LIN {X 0,Y 411.201,Z 268.89,A -85,B 0,C 180,E1 -10404.471,E2 -10404.471} C_VEL
LIN {X 0,Y 411.211,Z 268.89,A -85,B 0,C 180,E1 -10406.873,E2 -10406.873} C_VEL
LIN {X 0,Y 411.237,Z 268.886,A -85,B 0,C 180,E1 -10410.644,E2 -10410.644} C_VEL
LIN {X 0,Y 411.238,Z 268.882,A -85,B 0,C 180,E1 -10413.619,E2 -10413.619} C_VEL
LIN {X 0,Y 411.2,Z 268.891,A -85,B 0,C 180,E1 -10416.852,E2 -10416.852} C_VEL
LIN {X 0,Y 411.219,Z 268.887,A -85,B 0,C 180,E1 -10420.05,E2 -10420.05} C_VEL
LIN {X 0,Y 411.268,Z 268.88,A -85,B 0,C 180,E1 -10423.131,E2 -10423.131} C_VEL
LIN {X 0,Y 411.31,Z 268.874,A -85,B 0,C 180,E1 -10426.896,E2 -10426.896} C_VEL
LIN {X 0,Y 411.296,Z 268.879,A -85,B 0,C 180,E1 -10430.161,E2 -10430.161} C_VEL
LIN {X 0,Y 411.395,Z 268.863,A -85,B 0,C 180,E1 -10433.132,E2 -10433.132} C_VEL
LIN {X 0,Y 411.302,Z 268.875,A -85,B 0,C 180,E1 -10435.099,E2 -10435.099} C_VEL
LIN {X 0,Y 411.515,Z 268.851,A -85,B 0,C 180,E1 -10438.042,E2 -10438.042} C_VEL
LIN {X 0,Y 411.638,Z 268.837,A -85,B 0,C 180,E1 -10440,E2 -10440} C_VEL
LIN {X 0,Y 411.462,Z 268.856,A -85,B 0,C 180,E1 -10442.937,E2 -10442.937} C_VEL
LIN {X 0,Y 411.441,Z 268.861,A -85,B 0,C 180,E1 -10445.882,E2 -10445.882} C_VEL
LIN {X 0,Y 411.321,Z 268.872,A -85,B 0,C 180,E1 -10448.846,E2 -10448.846} C_VEL
LIN {X 0,Y 411.287,Z 268.88,A -85,B 0,C 180,E1 -10451.832,E2 -10451.832} C_VEL
LIN {X 0,Y 411.262,Z 268.879,A -85,B 0,C 180,E1 -10454.852,E2 -10454.852} C_VEL
LIN {X 0,Y 411.254,Z 268.884,A -85,B 0,C 180,E1 -10457.915,E2 -10457.915} C_VEL
LIN {X 0,Y 411.2,Z 268.889,A -85,B 0,C 180,E1 -10461.034,E2 -10461.034} C_VEL
LIN {X 0,Y 411.221,Z 268.886,A -85,B 0,C 180,E1 -10464.216,E2 -10464.216} C_VEL
LIN {X 0,Y 411.181,Z 268.895,A -85,B 0,C 180,E1 -10467.483,E2 -10467.483} C_VEL
LIN {X 0,Y 411.199,Z 268.89,A -85,B 0,C 180,E1 -10469.713,E2 -10469.713} C_VEL
LIN {X 0,Y 411.209,Z 268.89,A -85,B 0,C 180,E1 -10473.155,E2 -10473.155} C_VEL
LIN {X 0,Y 411.194,Z 268.889,A -85,B 0,C 180,E1 -10476.552,E2 -10476.552} C_VEL
LIN {X 0,Y 411.212,Z 268.897,A -85,B 0,C 180,E1 -10477.046,E2 -10477.046} C_VEL
LIN {X 0,Y 412.12,Z 274.033,A -85,B 0,C 180,E1 -10480.393,E2 -10480.393} C_VEL
LIN {X 0,Y 413.062,Z 279.177,A -85,B 0,C 180,E1 -10483.557,E2 -10483.557} C_VEL
LIN {X 0,Y 413.812,Z 283.108,A -85,B 0,C 180,E1 -10485.867,E2 -10485.867} C_VEL
LIN {X 0,Y 414.18,Z 285.575,A -85,B 0,C 180,E1 -10487.254,E2 -10487.254} C_VEL
LIN {X 0,Y 414.126,Z 289.23,A -85,B 0,C 180,E1 -10489.204,E2 -10489.204} C_VEL
LIN {X 0,Y 413.62,Z 295.329,A -85,B 0,C 180,E1 -10492.288,E2 -10492.288} C_VEL
LIN {X 0,Y 412.949,Z 302.639,A -85,B 0,C 180,E1 -10495.831,E2 -10495.831} C_VEL
LIN {X 0,Y 412.403,Z 309.967,A -85,B 0,C 180,E1 -10499.253,E2 -10499.253} C_VEL
LIN {X 0,Y 411.862,Z 317.318,A -85,B 0,C 180,E1 -10502.566,E2 -10502.566} C_VEL
LIN {X 0,Y 411.503,Z 322.706,A -85,B 0,C 180,E1 -10504.939,E2 -10504.939} C_VEL
LIN {X 0,Y 416.225,Z 340.747,A -85,B 0,C 180,E1 -10505.754,E2 -10505.754} C_VEL
LIN {X 0,Y 419.587,Z 356.286,A -85,B 0,C 180,E1 -10506.607,E2 -10506.607} C_VEL
LIN {X 0,Y 420.32,Z 360.595,A -85,B 0,C 180,E1 -10506.872,E2 -10506.872} C_VEL
LIN {X 0,Y 419.211,Z 375.514,A -85,B 0,C 180,E1 -10507.709,E2 -10507.709} C_VEL
LIN {X 0,Y 417.84,Z 389.213,A -85,B 0,C 180,E1 -10508.67,E2 -10508.67} C_VEL
LIN {X 0,Y 416.464,Z 403.182,A -85,B 0,C 180,E1 -10509.889,E2 -10509.889} C_VEL
LIN {X 0,Y 415.124,Z 415.883,A -85,B 0,C 180,E1 -10511.236,E2 -10511.236} C_VEL
LIN {X 0,Y 413.929,Z 427.487,A -85,B 0,C 180,E1 -10512.715,E2 -10512.715} C_VEL
LIN {X 0,Y 412.908,Z 437.298,A -85,B 0,C 180,E1 -10514.197,E2 -10514.197} C_VEL
LIN {X 0,Y 411.877,Z 446.94,A -85,B 0,C 180,E1 -10515.927,E2 -10515.927} C_VEL
LIN {X 0,Y 411.227,Z 455.004,A -85,B 0,C 180,E1 -10517.665,E2 -10517.665} C_VEL
LIN {X 0,Y 410.756,Z 460.8,A -85,B 0,C 180,E1 -10519.152,E2 -10519.152} C_VEL
LIN {X 0,Y 410.323,Z 467.138,A -85,B 0,C 180,E1 -10521.132,E2 -10521.132} C_VEL
LIN {X 0,Y 410.085,Z 472.043,A -85,B 0,C 180,E1 -10523.11,E2 -10523.11} C_VEL
LIN {X 0,Y 409.996,Z 475.633,A -85,B 0,C 180,E1 -10525.083,E2 -10525.083} C_VEL
LIN {X 0,Y 409.969,Z 477.983,A -85,B 0,C 180,E1 -10527.052,E2 -10527.052} C_VEL
LIN {X 0,Y 409.915,Z 479.141,A -85,B 0,C 180,E1 -10529.018,E2 -10529.018} C_VEL
LIN {X 0,Y 409.915,Z 479.086,A -85,B 0,C 180,E1 -10530.982,E2 -10530.982} C_VEL
LIN {X 0,Y 409.985,Z 477.829,A -85,B 0,C 180,E1 -10532.948,E2 -10532.948} C_VEL
LIN {X 0,Y 410.028,Z 475.37,A -85,B 0,C 180,E1 -10534.916,E2 -10534.916} C_VEL
LIN {X 0,Y 410.157,Z 471.659,A -85,B 0,C 180,E1 -10536.889,E2 -10536.889} C_VEL
LIN {X 0,Y 410.323,Z 466.595,A -85,B 0,C 180,E1 -10538.868,E2 -10538.868} C_VEL
LIN {X 0,Y 410.753,Z 460.062,A -85,B 0,C 180,E1 -10540.848,E2 -10540.848} C_VEL
LIN {X 0,Y 411.305,Z 451.879,A -85,B 0,C 180,E1 -10542.834,E2 -10542.834} C_VEL
LIN {X 0,Y 412.101,Z 443.193,A -85,B 0,C 180,E1 -10544.569,E2 -10544.569} C_VEL
LIN {X 0,Y 413.088,Z 432.798,A -85,B 0,C 180,E1 -10546.303,E2 -10546.303} C_VEL
LIN {X 0,Y 414.152,Z 422.254,A -85,B 0,C 180,E1 -10547.786,E2 -10547.786} C_VEL
LIN {X 0,Y 415.43,Z 409.781,A -85,B 0,C 180,E1 -10549.262,E2 -10549.262} C_VEL
LIN {X 0,Y 416.906,Z 396.092,A -85,B 0,C 180,E1 -10550.604,E2 -10550.604} C_VEL
LIN {X 0,Y 418.219,Z 382.713,A -85,B 0,C 180,E1 -10551.697,E2 -10551.697} C_VEL
LIN {X 0,Y 419.634,Z 367.281,A -85,B 0,C 180,E1 -10552.719,E2 -10552.719} C_VEL
LIN {X 0,Y 420.195,Z 359.819,A -85,B 0,C 180,E1 -10553.139,E2 -10553.139} C_VEL
LIN {X 0,Y 416.862,Z 341.94,A -85,B 0,C 180,E1 -10554.264,E2 -10554.264} C_VEL
LIN {X 0,Y 413.724,Z 327.801,A -85,B 0,C 180,E1 -10555.054,E2 -10555.054} C_VEL
LIN {X 0,Y 411.367,Z 319.22,A -85,B 0,C 180,E1 -10555.531,E2 -10555.531} C_VEL
LIN {X 0,Y 411.324,Z 318.857,A -85,B 0,C 180,E1 -10555.558,E2 -10555.558} C_VEL
LIN {X 0,Y 411.791,Z 310.923,A -85,B 0,C 180,E1 -10559.035,E2 -10559.035} C_VEL
LIN {X 0,Y 412.204,Z 304.79,A -85,B 0,C 180,E1 -10561.907,E2 -10561.907} C_VEL
LIN {X 0,Y 412.598,Z 300.233,A -85,B 0,C 180,E1 -10564.202,E2 -10564.202} C_VEL
LIN {X 0,Y 413.181,Z 295.3,A -85,B 0,C 180,E1 -10566.923,E2 -10566.923} C_VEL
LIN {X 0,Y 413.606,Z 292.035,A -85,B 0,C 180,E1 -10568.955,E2 -10568.955} C_VEL
LIN {X 0,Y 414.122,Z 288.293,A -85,B 0,C 180,E1 -10571.693,E2 -10571.693} C_VEL
LIN {X 0,Y 414.188,Z 286.686,A -85,B 0,C 180,E1 -10573.145,E2 -10573.145} C_VEL
LIN {X 0,Y 413.862,Z 284.426,A -85,B 0,C 180,E1 -10575.874,E2 -10575.874} C_VEL
LIN {X 0,Y 413.339,Z 283.119,A -85,B 0,C 180,E1 -10578.462,E2 -10578.462} C_VEL
LIN {X 0,Y 412.687,Z 282.48,A -85,B 0,C 180,E1 -10581.571,E2 -10581.571} C_VEL
LIN {X 0,Y 412.117,Z 282.678,A -85,B 0,C 180,E1 -10584.942,E2 -10584.942} C_VEL
LIN {X 0,Y 411.744,Z 283.465,A -85,B 0,C 180,E1 -10588.053,E2 -10588.053} C_VEL
LIN {X 0,Y 411.505,Z 284.692,A -85,B 0,C 180,E1 -10590.943,E2 -10590.943} C_VEL
LIN {X 0,Y 412.791,Z 287.703,A -85,B 0,C 180,E1 -10591.185,E2 -10591.185} C_VEL
LIN {X 0,Y 417.521,Z 298.226,A -85,B 0,C 180,E1 -10592.052,E2 -10592.052} C_VEL
LIN {X 0,Y 420.696,Z 307.253,A -85,B 0,C 180,E1 -10592.755,E2 -10592.755} C_VEL
LIN {X 0,Y 421.109,Z 308.983,A -85,B 0,C 180,E1 -10592.883,E2 -10592.883} C_VEL
LIN {X 0,Y 419.888,Z 325.497,A -85,B 0,C 180,E1 -10593.81,E2 -10593.81} C_VEL
LIN {X 0,Y 418.719,Z 339.594,A -85,B 0,C 180,E1 -10594.806,E2 -10594.806} C_VEL
LIN {X 0,Y 417.353,Z 353.955,A -85,B 0,C 180,E1 -10596.05,E2 -10596.05} C_VEL
LIN {X 0,Y 416.141,Z 366.806,A -85,B 0,C 180,E1 -10597.405,E2 -10597.405} C_VEL
LIN {X 0,Y 414.952,Z 378.132,A -85,B 0,C 180,E1 -10598.834,E2 -10598.834} C_VEL
LIN {X 0,Y 413.87,Z 388.594,A -85,B 0,C 180,E1 -10600.405,E2 -10600.405} C_VEL
LIN {X 0,Y 412.815,Z 398.291,A -85,B 0,C 180,E1 -10602.155,E2 -10602.155} C_VEL
LIN {X 0,Y 412.033,Z 406.284,A -85,B 0,C 180,E1 -10603.909,E2 -10603.909} C_VEL
LIN {X 0,Y 411.408,Z 412.88,A -85,B 0,C 180,E1 -10605.659,E2 -10605.659} C_VEL
LIN {X 0,Y 410.912,Z 418.826,A -85,B 0,C 180,E1 -10607.656,E2 -10607.656} C_VEL
LIN {X 0,Y 410.554,Z 422.279,A -85,B 0,C 180,E1 -10609.147,E2 -10609.147} C_VEL
LIN {X 0,Y 410.316,Z 425.719,A -85,B 0,C 180,E1 -10611.132,E2 -10611.132} C_VEL
LIN {X 0,Y 410.238,Z 427.874,A -85,B 0,C 180,E1 -10613.113,E2 -10613.113} C_VEL
LIN {X 0,Y 410.113,Z 428.803,A -85,B 0,C 180,E1 -10615.085,E2 -10615.085} C_VEL
LIN {X 0,Y 410.182,Z 428.514,A -85,B 0,C 180,E1 -10617.054,E2 -10617.054} C_VEL
LIN {X 0,Y 410.116,Z 427.022,A -85,B 0,C 180,E1 -10619.018,E2 -10619.018} C_VEL
LIN {X 0,Y 410.165,Z 424.281,A -85,B 0,C 180,E1 -10620.982,E2 -10620.982} C_VEL
LIN {X 0,Y 410.423,Z 420.261,A -85,B 0,C 180,E1 -10622.945,E2 -10622.945} C_VEL
LIN {X 0,Y 410.871,Z 414.887,A -85,B 0,C 180,E1 -10624.906,E2 -10624.906} C_VEL
LIN {X 0,Y 411.131,Z 408.051,A -85,B 0,C 180,E1 -10626.873,E2 -10626.873} C_VEL
LIN {X 0,Y 411.783,Z 400.661,A -85,B 0,C 180,E1 -10628.589,E2 -10628.589} C_VEL
LIN {X 0,Y 412.563,Z 391.796,A -85,B 0,C 180,E1 -10630.304,E2 -10630.304} C_VEL
LIN {X 0,Y 413.371,Z 382.811,A -85,B 0,C 180,E1 -10631.772,E2 -10631.772} C_VEL
LIN {X 0,Y 414.331,Z 372.247,A -85,B 0,C 180,E1 -10633.238,E2 -10633.238} C_VEL
LIN {X 0,Y 415.304,Z 360.819,A -85,B 0,C 180,E1 -10634.58,E2 -10634.58} C_VEL
LIN {X 0,Y 416.359,Z 347.121,A -85,B 0,C 180,E1 -10635.92,E2 -10635.92} C_VEL
LIN {X 0,Y 417.483,Z 333.527,A -85,B 0,C 180,E1 -10637.008,E2 -10637.008} C_VEL
LIN {X 0,Y 418.43,Z 319.094,A -85,B 0,C 180,E1 -10637.948,E2 -10637.948} C_VEL
LIN {X 0,Y 419.125,Z 307.156,A -85,B 0,C 180,E1 -10638.578,E2 -10638.578} C_VEL
LIN {X 0,Y 415.577,Z 293.478,A -85,B 0,C 180,E1 -10639.353,E2 -10639.353} C_VEL
LIN {X 0,Y 410.491,Z 277.04,A -85,B 0,C 180,E1 -10640.132,E2 -10640.132} C_VEL
LIN {X 0,Y 410.369,Z 276.211,A -85,B 0,C 180,E1 -10640.163,E2 -10640.163} C_VEL
LIN {X 0,Y 410.377,Z 273.314,A -85,B 0,C 180,E1 -10643.197,E2 -10643.197} C_VEL
LIN {X 0,Y 410.444,Z 271.32,A -85,B 0,C 180,E1 -10645.346,E2 -10645.346} C_VEL
LIN {X 0,Y 410.452,Z 269.277,A -85,B 0,C 180,E1 -10647.537,E2 -10647.537} C_VEL
LIN {X 0,Y 410.683,Z 268.956,A -85,B 0,C 180,E1 -10649.754,E2 -10649.754} C_VEL
LIN {X 0,Y 411.018,Z 268.915,A -85,B 0,C 180,E1 -10653.085,E2 -10653.085} C_VEL
LIN {X 0,Y 411.15,Z 268.896,A -85,B 0,C 180,E1 -10655.534,E2 -10655.534} C_VEL
LIN {X 0,Y 411.202,Z 268.887,A -85,B 0,C 180,E1 -10658.168,E2 -10658.168} C_VEL
LIN {X 0,Y 411.164,Z 268.896,A -85,B 0,C 180,E1 -10661.228,E2 -10661.228} C_VEL
LIN {X 0,Y 411.179,Z 268.891,A -85,B 0,C 180,E1 -10664.49,E2 -10664.49} C_VEL
LIN {X 0,Y 411.181,Z 268.892,A -85,B 0,C 180,E1 -10668.195,E2 -10668.195} C_VEL
LIN {X 0,Y 411.217,Z 268.89,A -85,B 0,C 180,E1 -10670.775,E2 -10670.775} C_VEL
LIN {X 0,Y 411.2,Z 268.891,A -85,B 0,C 180,E1 -10674.471,E2 -10674.471} C_VEL
LIN {X 0,Y 411.21,Z 268.89,A -85,B 0,C 180,E1 -10676.873,E2 -10676.873} C_VEL
LIN {X 0,Y 411.236,Z 268.886,A -85,B 0,C 180,E1 -10680.644,E2 -10680.644} C_VEL
LIN {X 0,Y 411.236,Z 268.883,A -85,B 0,C 180,E1 -10683.619,E2 -10683.619} C_VEL
LIN {X 0,Y 411.198,Z 268.89,A -85,B 0,C 180,E1 -10686.852,E2 -10686.852} C_VEL
LIN {X 0,Y 411.218,Z 268.887,A -85,B 0,C 180,E1 -10690.051,E2 -10690.051} C_VEL
LIN {X 0,Y 411.266,Z 268.88,A -85,B 0,C 180,E1 -10693.131,E2 -10693.131} C_VEL
LIN {X 0,Y 411.309,Z 268.875,A -85,B 0,C 180,E1 -10696.896,E2 -10696.896} C_VEL
LIN {X 0,Y 411.295,Z 268.879,A -85,B 0,C 180,E1 -10700.161,E2 -10700.161} C_VEL
LIN {X 0,Y 411.395,Z 268.864,A -85,B 0,C 180,E1 -10703.132,E2 -10703.132} C_VEL
LIN {X 0,Y 411.3,Z 268.874,A -85,B 0,C 180,E1 -10705.099,E2 -10705.099} C_VEL
LIN {X 0,Y 411.513,Z 268.851,A -85,B 0,C 180,E1 -10708.043,E2 -10708.043} C_VEL
LIN {X 0,Y 411.639,Z 268.836,A -85,B 0,C 180,E1 -10710,E2 -10710} C_VEL
LIN {X 0,Y 411.453,Z 268.856,A -85,B 0,C 180,E1 -10712.937,E2 -10712.937} C_VEL
LIN {X 0,Y 411.428,Z 268.86,A -85,B 0,C 180,E1 -10716.868,E2 -10716.868} C_VEL
LIN {X 0,Y 411.294,Z 268.879,A -85,B 0,C 180,E1 -10719.839,E2 -10719.839} C_VEL
LIN {X 0,Y 411.283,Z 268.88,A -85,B 0,C 180,E1 -10721.772,E2 -10721.772} C_VEL
LIN {X 0,Y 410.639,Z 268.964,A -85,B 0,C 180,E1 -10722.589,E2 -10722.589} C_VEL
LIN {X 0,Y 407.748,Z 269.321,A -85,B 0,C 180,E1 -10723.915,E2 -10723.915} C_VEL
LIN {X 0,Y 405.304,Z 269.623,A -85,B 0,C 180,E1 -10724.987,E2 -10724.987} C_VEL
LIN {X 0,Y 404.285,Z 269.752,A -85,B 0,C 180,E1 -10725.816,E2 -10725.816} C_VEL
LIN {X 0,Y 404.22,Z 269.758,A -85,B 0,C 180,E1 -10726.097,E2 -10726.097} C_VEL
LIN {X 0,Y 404.166,Z 269.767,A -85,B 0,C 180,E1 -10729.293,E2 -10729.293} C_VEL
LIN {X 0,Y 404.159,Z 269.764,A -85,B 0,C 180,E1 -10732.834,E2 -10732.834} C_VEL
LIN {X 0,Y 404.187,Z 269.765,A -85,B 0,C 180,E1 -10735.766,E2 -10735.766} C_VEL
LIN {X 0,Y 404.199,Z 269.76,A -85,B 0,C 180,E1 -10738,E2 -10738} C_VEL
LIN {X 0,Y 404.143,Z 269.769,A -85,B 0,C 180,E1 -10741.558,E2 -10741.558} C_VEL
LIN {X 0,Y 404.188,Z 269.764,A -85,B 0,C 180,E1 -10745.016,E2 -10745.016} C_VEL
LIN {X 0,Y 404.139,Z 269.771,A -85,B 0,C 180,E1 -10748.759,E2 -10748.759} C_VEL
LIN {X 0,Y 404.111,Z 269.772,A -85,B 0,C 180,E1 -10751.597,E2 -10751.597} C_VEL
LIN {X 0,Y 404.147,Z 269.768,A -85,B 0,C 180,E1 -10754.522,E2 -10754.522} C_VEL
LIN {X 0,Y 404.14,Z 269.77,A -85,B 0,C 180,E1 -10757.296,E2 -10757.296} C_VEL
LIN {X 0,Y 404.173,Z 269.762,A -85,B 0,C 180,E1 -10759.955,E2 -10759.955} C_VEL
LIN {X 0,Y 404.14,Z 269.77,A -85,B 0,C 180,E1 -10763.125,E2 -10763.125} C_VEL
LIN {X 0,Y 404.148,Z 269.767,A -85,B 0,C 180,E1 -10766.188,E2 -10766.188} C_VEL
LIN {X 0,Y 404.15,Z 269.766,A -85,B 0,C 180,E1 -10769.715,E2 -10769.715} C_VEL
LIN {X 0,Y 404.197,Z 269.76,A -85,B 0,C 180,E1 -10773.123,E2 -10773.123} C_VEL
LIN {X 0,Y 404.174,Z 269.763,A -85,B 0,C 180,E1 -10775.334,E2 -10775.334} C_VEL
LIN {X 0,Y 404.143,Z 269.771,A -85,B 0,C 180,E1 -10778.581,E2 -10778.581} C_VEL
LIN {X 0,Y 404.213,Z 269.759,A -85,B 0,C 180,E1 -10781.762,E2 -10781.762} C_VEL
LIN {X 0,Y 404.209,Z 269.76,A -85,B 0,C 180,E1 -10784.882,E2 -10784.882} C_VEL
LIN {X 0,Y 404.261,Z 269.754,A -85,B 0,C 180,E1 -10787.958,E2 -10787.958} C_VEL
LIN {X 0,Y 404.27,Z 269.752,A -85,B 0,C 180,E1 -10790.998,E2 -10790.998} C_VEL
LIN {X 0,Y 404.382,Z 269.741,A -85,B 0,C 180,E1 -10794.014,E2 -10794.014} C_VEL
LIN {X 0,Y 404.483,Z 269.727,A -85,B 0,C 180,E1 -10798.008,E2 -10798.008} C_VEL
LIN {X 0,Y 404.607,Z 269.713,A -85,B 0,C 180,E1 -10800,E2 -10800} C_VEL
LIN {X 0,Y 404.42,Z 269.733,A -85,B 0,C 180,E1 -10802.988,E2 -10802.988} C_VEL
LIN {X 0,Y 404.388,Z 269.74,A -85,B 0,C 180,E1 -10805.985,E2 -10805.985} C_VEL
LIN {X 0,Y 404.268,Z 269.751,A -85,B 0,C 180,E1 -10809.001,E2 -10809.001} C_VEL
LIN {X 0,Y 404.26,Z 269.756,A -85,B 0,C 180,E1 -10812.041,E2 -10812.041} C_VEL
LIN {X 0,Y 404.209,Z 269.759,A -85,B 0,C 180,E1 -10815.118,E2 -10815.118} C_VEL
LIN {X 0,Y 404.212,Z 269.76,A -85,B 0,C 180,E1 -10818.238,E2 -10818.238} C_VEL
LIN {X 0,Y 404.163,Z 269.768,A -85,B 0,C 180,E1 -10821.418,E2 -10821.418} C_VEL
LIN {X 0,Y 404.169,Z 269.764,A -85,B 0,C 180,E1 -10824.666,E2 -10824.666} C_VEL
LIN {X 0,Y 404.122,Z 269.769,A -85,B 0,C 180,E1 -10828.005,E2 -10828.005} C_VEL
LIN {X 0,Y 404.146,Z 269.768,A -85,B 0,C 180,E1 -10830.285,E2 -10830.285} C_VEL
LIN {X 0,Y 404.147,Z 269.77,A -85,B 0,C 180,E1 -10833.812,E2 -10833.812} C_VEL
LIN {X 0,Y 404.173,Z 269.783,A -85,B 0,C 180,E1 -10836.573,E2 -10836.573} C_VEL
LIN {X 0,Y 405.142,Z 275.313,A -85,B 0,C 180,E1 -10840.246,E2 -10840.246} C_VEL
LIN {X 0,Y 406.053,Z 280.309,A -85,B 0,C 180,E1 -10843.369,E2 -10843.369} C_VEL
LIN {X 0,Y 407.006,Z 285.588,A -85,B 0,C 180,E1 -10846.488,E2 -10846.488} C_VEL
LIN {X 0,Y 407.238,Z 289.15,A -85,B 0,C 180,E1 -10848.465,E2 -10848.465} C_VEL
LIN {X 0,Y 406.752,Z 295.053,A -85,B 0,C 180,E1 -10851.536,E2 -10851.536} C_VEL
LIN {X 0,Y 406.18,Z 300.831,A -85,B 0,C 180,E1 -10854.412,E2 -10854.412} C_VEL
LIN {X 0,Y 405.634,Z 307.255,A -85,B 0,C 180,E1 -10857.513,E2 -10857.513} C_VEL
LIN {X 0,Y 405.08,Z 314.592,A -85,B 0,C 180,E1 -10860.935,E2 -10860.935} C_VEL
LIN {X 0,Y 404.491,Z 322.42,A -85,B 0,C 180,E1 -10864.471,E2 -10864.471} C_VEL
LIN {X 0,Y 409.547,Z 341.563,A -85,B 0,C 180,E1 -10865.375,E2 -10865.375} C_VEL
LIN {X 0,Y 412.792,Z 356.751,A -85,B 0,C 180,E1 -10866.243,E2 -10866.243} C_VEL
LIN {X 0,Y 413.652,Z 361.682,A -85,B 0,C 180,E1 -10866.558,E2 -10866.558} C_VEL
LIN {X 0,Y 412.586,Z 375.074,A -85,B 0,C 180,E1 -10867.332,E2 -10867.332} C_VEL
LIN {X 0,Y 411.174,Z 388.756,A -85,B 0,C 180,E1 -10868.307,E2 -10868.307} C_VEL
LIN {X 0,Y 409.711,Z 402.72,A -85,B 0,C 180,E1 -10869.543,E2 -10869.543} C_VEL
LIN {X 0,Y 408.321,Z 415.427,A -85,B 0,C 180,E1 -10870.911,E2 -10870.911} C_VEL
LIN {X 0,Y 407.091,Z 427.043,A -85,B 0,C 180,E1 -10872.415,E2 -10872.415} C_VEL
LIN {X 0,Y 405.964,Z 436.863,A -85,B 0,C 180,E1 -10873.919,E2 -10873.919} C_VEL
LIN {X 0,Y 404.913,Z 446.515,A -85,B 0,C 180,E1 -10875.68,E2 -10875.68} C_VEL
LIN {X 0,Y 404.214,Z 454.586,A -85,B 0,C 180,E1 -10877.447,E2 -10877.447} C_VEL
LIN {X 0,Y 403.565,Z 462.118,A -85,B 0,C 180,E1 -10879.464,E2 -10879.464} C_VEL
LIN {X 0,Y 403.177,Z 468.102,A -85,B 0,C 180,E1 -10881.479,E2 -10881.479} C_VEL
LIN {X 0,Y 403.028,Z 471.645,A -85,B 0,C 180,E1 -10882.989,E2 -10882.989} C_VEL
LIN {X 0,Y 402.907,Z 475.238,A -85,B 0,C 180,E1 -10884.996,E2 -10884.996} C_VEL
LIN {X 0,Y 402.869,Z 477.589,A -85,B 0,C 180,E1 -10887,E2 -10887} C_VEL
LIN {X 0,Y 402.844,Z 478.744,A -85,B 0,C 180,E1 -10889,E2 -10889} C_VEL
LIN {X 0,Y 402.844,Z 478.68,A -85,B 0,C 180,E1 -10891,E2 -10891} C_VEL
LIN {X 0,Y 402.885,Z 477.405,A -85,B 0,C 180,E1 -10893,E2 -10893} C_VEL
LIN {X 0,Y 402.939,Z 474.924,A -85,B 0,C 180,E1 -10895.003,E2 -10895.003} C_VEL
LIN {X 0,Y 403.067,Z 471.191,A -85,B 0,C 180,E1 -10897.011,E2 -10897.011} C_VEL
LIN {X 0,Y 403.264,Z 466.108,A -85,B 0,C 180,E1 -10899.024,E2 -10899.024} C_VEL
LIN {X 0,Y 403.705,Z 459.548,A -85,B 0,C 180,E1 -10901.04,E2 -10901.04} C_VEL
LIN {X 0,Y 404.301,Z 451.354,A -85,B 0,C 180,E1 -10903.061,E2 -10903.061} C_VEL
LIN {X 0,Y 405.141,Z 442.671,A -85,B 0,C 180,E1 -10904.825,E2 -10904.825} C_VEL
LIN {X 0,Y 406.171,Z 432.288,A -85,B 0,C 180,E1 -10906.589,E2 -10906.589} C_VEL
LIN {X 0,Y 407.299,Z 421.783,A -85,B 0,C 180,E1 -10908.095,E2 -10908.095} C_VEL
LIN {X 0,Y 408.65,Z 409.385,A -85,B 0,C 180,E1 -10909.595,E2 -10909.595} C_VEL
LIN {X 0,Y 410.217,Z 395.821,A -85,B 0,C 180,E1 -10910.955,E2 -10910.955} C_VEL
LIN {X 0,Y 411.606,Z 382.637,A -85,B 0,C 180,E1 -10912.064,E2 -10912.064} C_VEL
LIN {X 0,Y 413,Z 368.511,A -85,B 0,C 180,E1 -10913.041,E2 -10913.041} C_VEL
LIN {X 0,Y 413.608,Z 361.117,A -85,B 0,C 180,E1 -10913.482,E2 -10913.482} C_VEL
LIN {X 0,Y 410.285,Z 342.41,A -85,B 0,C 180,E1 -10914.726,E2 -10914.726} C_VEL
LIN {X 0,Y 407.411,Z 328.898,A -85,B 0,C 180,E1 -10915.538,E2 -10915.538} C_VEL
LIN {X 0,Y 404.84,Z 320.552,A -85,B 0,C 180,E1 -10916.066,E2 -10916.066} C_VEL
LIN {X 0,Y 404.332,Z 318.102,A -85,B 0,C 180,E1 -10916.206,E2 -10916.206} C_VEL
LIN {X 0,Y 404.916,Z 310.206,A -85,B 0,C 180,E1 -10919.792,E2 -10919.792} C_VEL
LIN {X 0,Y 405.535,Z 302.329,A -85,B 0,C 180,E1 -10923.711,E2 -10923.711} C_VEL
LIN {X 0,Y 406.252,Z 296.033,A -85,B 0,C 180,E1 -10927.271,E2 -10927.271} C_VEL
LIN {X 0,Y 406.778,Z 292.297,A -85,B 0,C 180,E1 -10929.737,E2 -10929.737} C_VEL
LIN {X 0,Y 407.218,Z 289.06,A -85,B 0,C 180,E1 -10932.306,E2 -10932.306} C_VEL
LIN {X 0,Y 407.211,Z 287.683,A -85,B 0,C 180,E1 -10933.659,E2 -10933.659} C_VEL
LIN {X 0,Y 406.843,Z 285.681,A -85,B 0,C 180,E1 -10936.293,E2 -10936.293} C_VEL
LIN {X 0,Y 406.271,Z 284.486,A -85,B 0,C 180,E1 -10938.902,E2 -10938.902} C_VEL
LIN {X 0,Y 405.77,Z 283.963,A -85,B 0,C 180,E1 -10941.426,E2 -10941.426} C_VEL
LIN {X 0,Y 405.205,Z 284.029,A -85,B 0,C 180,E1 -10944.606,E2 -10944.606} C_VEL
LIN {X 0,Y 404.841,Z 284.608,A -85,B 0,C 180,E1 -10947.442,E2 -10947.442} C_VEL
LIN {X 0,Y 404.584,Z 285.6,A -85,B 0,C 180,E1 -10950.291,E2 -10950.291} C_VEL
LIN {X 0,Y 405.759,Z 288.529,A -85,B 0,C 180,E1 -10950.534,E2 -10950.534} C_VEL
LIN {X 0,Y 410.274,Z 297.796,A -85,B 0,C 180,E1 -10951.391,E2 -10951.391} C_VEL
LIN {X 0,Y 414.47,Z 309.455,A -85,B 0,C 180,E1 -10952.373,E2 -10952.373} C_VEL
LIN {X 0,Y 414.688,Z 313.036,A -85,B 0,C 180,E1 -10952.594,E2 -10952.594} C_VEL
LIN {X 0,Y 413.419,Z 328.367,A -85,B 0,C 180,E1 -10953.512,E2 -10953.512} C_VEL
LIN {X 0,Y 412.038,Z 343.253,A -85,B 0,C 180,E1 -10954.638,E2 -10954.638} C_VEL
LIN {X 0,Y 410.659,Z 356.841,A -85,B 0,C 180,E1 -10955.884,E2 -10955.884} C_VEL
LIN {X 0,Y 409.346,Z 369.356,A -85,B 0,C 180,E1 -10957.276,E2 -10957.276} C_VEL
LIN {X 0,Y 408.021,Z 380.864,A -85,B 0,C 180,E1 -10958.795,E2 -10958.795} C_VEL
LIN {X 0,Y 406.973,Z 390.523,A -85,B 0,C 180,E1 -10960.322,E2 -10960.322} C_VEL
LIN {X 0,Y 405.883,Z 399.814,A -85,B 0,C 180,E1 -10962.068,E2 -10962.068} C_VEL
LIN {X 0,Y 405.056,Z 407.763,A -85,B 0,C 180,E1 -10963.883,E2 -10963.883} C_VEL
LIN {X 0,Y 404.307,Z 414.939,A -85,B 0,C 180,E1 -10965.915,E2 -10965.915} C_VEL
LIN {X 0,Y 403.8,Z 420.527,A -85,B 0,C 180,E1 -10967.945,E2 -10967.945} C_VEL
LIN {X 0,Y 403.401,Z 424.658,A -85,B 0,C 180,E1 -10969.967,E2 -10969.967} C_VEL
LIN {X 0,Y 403.201,Z 427.447,A -85,B 0,C 180,E1 -10971.985,E2 -10971.985} C_VEL
LIN {X 0,Y 403.154,Z 428.98,A -85,B 0,C 180,E1 -10973.996,E2 -10973.996} C_VEL
LIN {X 0,Y 403.053,Z 429.308,A -85,B 0,C 180,E1 -10976.001,E2 -10976.001} C_VEL
LIN {X 0,Y 403.07,Z 428.413,A -85,B 0,C 180,E1 -10978.002,E2 -10978.002} C_VEL
LIN {X 0,Y 403.034,Z 426.284,A -85,B 0,C 180,E1 -10980,E2 -10980} C_VEL
LIN {X 0,Y 403.183,Z 422.896,A -85,B 0,C 180,E1 -10981.998,E2 -10981.998} C_VEL
LIN {X 0,Y 403.614,Z 418.188,A -85,B 0,C 180,E1 -10983.994,E2 -10983.994} C_VEL
LIN {X 0,Y 403.939,Z 412.082,A -85,B 0,C 180,E1 -10985.992,E2 -10985.992} C_VEL
LIN {X 0,Y 404.486,Z 404.395,A -85,B 0,C 180,E1 -10987.99,E2 -10987.99} C_VEL
LIN {X 0,Y 405.199,Z 396.163,A -85,B 0,C 180,E1 -10989.736,E2 -10989.736} C_VEL
LIN {X 0,Y 406.159,Z 386.298,A -85,B 0,C 180,E1 -10991.478,E2 -10991.478} C_VEL
LIN {X 0,Y 407.008,Z 376.253,A -85,B 0,C 180,E1 -10992.972,E2 -10992.972} C_VEL
LIN {X 0,Y 408.141,Z 364.365,A -85,B 0,C 180,E1 -10994.459,E2 -10994.459} C_VEL
LIN {X 0,Y 409.285,Z 351.253,A -85,B 0,C 180,E1 -10995.828,E2 -10995.828} C_VEL
LIN {X 0,Y 410.32,Z 338.552,A -85,B 0,C 180,E1 -10996.929,E2 -10996.929} C_VEL
LIN {X 0,Y 411.324,Z 324.793,A -85,B 0,C 180,E1 -10997.912,E2 -10997.912} C_VEL
LIN {X 0,Y 412.32,Z 309.4,A -85,B 0,C 180,E1 -10998.787,E2 -10998.787} C_VEL
LIN {X 0,Y 411.736,Z 305.45,A -85,B 0,C 180,E1 -10999.017,E2 -10999.017} C_VEL
LIN {X 0,Y 407.389,Z 290.124,A -85,B 0,C 180,E1 -10999.885,E2 -10999.885} C_VEL
LIN {X 0,Y 403.303,Z 276.594,A -85,B 0,C 180,E1 -11000.53,E2 -11000.53} C_VEL
LIN {X 0,Y 403.354,Z 273.649,A -85,B 0,C 180,E1 -11003.625,E2 -11003.625} C_VEL
LIN {X 0,Y 403.399,Z 270.572,A -85,B 0,C 180,E1 -11006.935,E2 -11006.935} C_VEL
LIN {X 0,Y 403.421,Z 269.861,A -85,B 0,C 180,E1 -11008.058,E2 -11008.058} C_VEL
LIN {X 0,Y 403.826,Z 269.811,A -85,B 0,C 180,E1 -11011.474,E2 -11011.474} C_VEL
LIN {X 0,Y 404.107,Z 269.774,A -85,B 0,C 180,E1 -11015.024,E2 -11015.024} C_VEL
LIN {X 0,Y 404.151,Z 269.767,A -85,B 0,C 180,E1 -11018.507,E2 -11018.507} C_VEL
LIN {X 0,Y 404.122,Z 269.771,A -85,B 0,C 180,E1 -11021.599,E2 -11021.599} C_VEL
LIN {X 0,Y 404.148,Z 269.767,A -85,B 0,C 180,E1 -11024.522,E2 -11024.522} C_VEL
LIN {X 0,Y 404.14,Z 269.77,A -85,B 0,C 180,E1 -11027.296,E2 -11027.296} C_VEL
LIN {X 0,Y 404.172,Z 269.763,A -85,B 0,C 180,E1 -11029.955,E2 -11029.955} C_VEL
LIN {X 0,Y 404.139,Z 269.77,A -85,B 0,C 180,E1 -11033.125,E2 -11033.125} C_VEL
LIN {X 0,Y 404.147,Z 269.768,A -85,B 0,C 180,E1 -11036.188,E2 -11036.188} C_VEL
LIN {X 0,Y 404.149,Z 269.766,A -85,B 0,C 180,E1 -11039.715,E2 -11039.715} C_VEL
LIN {X 0,Y 404.196,Z 269.761,A -85,B 0,C 180,E1 -11043.123,E2 -11043.123} C_VEL
LIN {X 0,Y 404.173,Z 269.763,A -85,B 0,C 180,E1 -11045.334,E2 -11045.334} C_VEL
LIN {X 0,Y 404.141,Z 269.77,A -85,B 0,C 180,E1 -11048.581,E2 -11048.581} C_VEL
LIN {X 0,Y 404.211,Z 269.758,A -85,B 0,C 180,E1 -11051.762,E2 -11051.762} C_VEL
LIN {X 0,Y 404.209,Z 269.76,A -85,B 0,C 180,E1 -11054.882,E2 -11054.882} C_VEL
LIN {X 0,Y 404.259,Z 269.755,A -85,B 0,C 180,E1 -11057.959,E2 -11057.959} C_VEL
LIN {X 0,Y 404.292,Z 269.749,A -85,B 0,C 180,E1 -11060.999,E2 -11060.999} C_VEL
LIN {X 0,Y 404.382,Z 269.74,A -85,B 0,C 180,E1 -11064.014,E2 -11064.014} C_VEL
LIN {X 0,Y 404.482,Z 269.727,A -85,B 0,C 180,E1 -11068.009,E2 -11068.009} C_VEL
LIN {X 0,Y 404.608,Z 269.712,A -85,B 0,C 180,E1 -11070,E2 -11070} C_VEL
LIN {X 0,Y 404.412,Z 269.733,A -85,B 0,C 180,E1 -11072.989,E2 -11072.989} C_VEL
LIN {X 0,Y 404.373,Z 269.739,A -85,B 0,C 180,E1 -11076.988,E2 -11076.988} C_VEL
LIN {X 0,Y 404.259,Z 269.754,A -85,B 0,C 180,E1 -11080.012,E2 -11080.012} C_VEL
LIN {X 0,Y 404.27,Z 269.753,A -85,B 0,C 180,E1 -11083.211,E2 -11083.211} C_VEL
LIN {X 0,Y 404.22,Z 269.758,A -85,B 0,C 180,E1 -11086.097,E2 -11086.097} C_VEL
LIN {X 0,Y 403.604,Z 269.838,A -85,B 0,C 180,E1 -11086.928,E2 -11086.928} C_VEL
LIN {X 0,Y 400.767,Z 270.192,A -85,B 0,C 180,E1 -11088.279,E2 -11088.279} C_VEL
LIN {X 0,Y 398.314,Z 270.496,A -85,B 0,C 180,E1 -11089.37,E2 -11089.37} C_VEL
LIN {X 0,Y 397.227,Z 270.629,A -85,B 0,C 180,E1 -11090.213,E2 -11090.213} C_VEL
LIN {X 0,Y 397.122,Z 270.641,A -85,B 0,C 180,E1 -11090.5,E2 -11090.5} C_VEL
LIN {X 0,Y 397.136,Z 270.641,A -85,B 0,C 180,E1 -11094.018,E2 -11094.018} C_VEL
LIN {X 0,Y 397.198,Z 270.635,A -85,B 0,C 180,E1 -11097.39,E2 -11097.39} C_VEL
LIN {X 0,Y 397.082,Z 270.648,A -85,B 0,C 180,E1 -11100.882,E2 -11100.882} C_VEL
LIN {X 0,Y 397.129,Z 270.641,A -85,B 0,C 180,E1 -11104.493,E2 -11104.493} C_VEL
LIN {X 0,Y 397.096,Z 270.645,A -85,B 0,C 180,E1 -11108.276,E2 -11108.276} C_VEL
LIN {X 0,Y 397.055,Z 270.649,A -85,B 0,C 180,E1 -11111.977,E2 -11111.977} C_VEL
LIN {X 0,Y 397.09,Z 270.648,A -85,B 0,C 180,E1 -11115.069,E2 -11115.069} C_VEL
LIN {X 0,Y 397.07,Z 270.648,A -85,B 0,C 180,E1 -11118.021,E2 -11118.021} C_VEL
LIN {X 0,Y 397.135,Z 270.642,A -85,B 0,C 180,E1 -11121.138,E2 -11121.138} C_VEL
LIN {X 0,Y 397.123,Z 270.644,A -85,B 0,C 180,E1 -11124.497,E2 -11124.497} C_VEL
LIN {X 0,Y 397.082,Z 270.646,A -85,B 0,C 180,E1 -11127.928,E2 -11127.928} C_VEL
LIN {X 0,Y 397.126,Z 270.641,A -85,B 0,C 180,E1 -11131.456,E2 -11131.456} C_VEL
LIN {X 0,Y 397.155,Z 270.642,A -85,B 0,C 180,E1 -11134.488,E2 -11134.488} C_VEL
LIN {X 0,Y 397.1,Z 270.647,A -85,B 0,C 180,E1 -11138.181,E2 -11138.181} C_VEL
LIN {X 0,Y 397.165,Z 270.635,A -85,B 0,C 180,E1 -11141.426,E2 -11141.426} C_VEL
LIN {X 0,Y 397.183,Z 270.638,A -85,B 0,C 180,E1 -11144.608,E2 -11144.608} C_VEL
LIN {X 0,Y 397.224,Z 270.629,A -85,B 0,C 180,E1 -11147.742,E2 -11147.742} C_VEL
LIN {X 0,Y 397.24,Z 270.628,A -85,B 0,C 180,E1 -11150.838,E2 -11150.838} C_VEL
LIN {X 0,Y 397.333,Z 270.618,A -85,B 0,C 180,E1 -11153.908,E2 -11153.908} C_VEL
LIN {X 0,Y 397.452,Z 270.603,A -85,B 0,C 180,E1 -11157.973,E2 -11157.973} C_VEL
LIN {X 0,Y 397.577,Z 270.589,A -85,B 0,C 180,E1 -11160,E2 -11160} C_VEL
LIN {X 0,Y 397.379,Z 270.609,A -85,B 0,C 180,E1 -11163.041,E2 -11163.041} C_VEL
LIN {X 0,Y 397.338,Z 270.618,A -85,B 0,C 180,E1 -11166.092,E2 -11166.092} C_VEL
LIN {X 0,Y 397.238,Z 270.627,A -85,B 0,C 180,E1 -11169.162,E2 -11169.162} C_VEL
LIN {X 0,Y 397.223,Z 270.631,A -85,B 0,C 180,E1 -11172.258,E2 -11172.258} C_VEL
LIN {X 0,Y 397.182,Z 270.636,A -85,B 0,C 180,E1 -11175.392,E2 -11175.392} C_VEL
LIN {X 0,Y 397.164,Z 270.636,A -85,B 0,C 180,E1 -11178.573,E2 -11178.573} C_VEL
LIN {X 0,Y 397.112,Z 270.645,A -85,B 0,C 180,E1 -11181.817,E2 -11181.817} C_VEL
LIN {X 0,Y 397.111,Z 270.646,A -85,B 0,C 180,E1 -11185.134,E2 -11185.134} C_VEL
LIN {X 0,Y 397.074,Z 270.647,A -85,B 0,C 180,E1 -11188.547,E2 -11188.547} C_VEL
LIN {X 0,Y 397.084,Z 270.649,A -85,B 0,C 180,E1 -11191.836,E2 -11191.836} C_VEL
LIN {X 0,Y 397.127,Z 270.643,A -85,B 0,C 180,E1 -11194.493,E2 -11194.493} C_VEL
LIN {X 0,Y 397.141,Z 270.811,A -85,B 0,C 180,E1 -11196.201,E2 -11196.201} C_VEL
LIN {X 0,Y 397.985,Z 275.628,A -85,B 0,C 180,E1 -11199.473,E2 -11199.473} C_VEL
LIN {X 0,Y 398.825,Z 279.942,A -85,B 0,C 180,E1 -11202.258,E2 -11202.258} C_VEL
LIN {X 0,Y 399.956,Z 286.257,A -85,B 0,C 180,E1 -11206.091,E2 -11206.091} C_VEL
LIN {X 0,Y 400.262,Z 289.872,A -85,B 0,C 180,E1 -11208.147,E2 -11208.147} C_VEL
LIN {X 0,Y 399.885,Z 294.765,A -85,B 0,C 180,E1 -11210.75,E2 -11210.75} C_VEL
LIN {X 0,Y 399.414,Z 299.635,A -85,B 0,C 180,E1 -11213.254,E2 -11213.254} C_VEL
LIN {X 0,Y 398.703,Z 306.967,A -85,B 0,C 180,E1 -11216.876,E2 -11216.876} C_VEL
LIN {X 0,Y 398.116,Z 314.299,A -85,B 0,C 180,E1 -11220.377,E2 -11220.377} C_VEL
LIN {X 0,Y 397.553,Z 321.629,A -85,B 0,C 180,E1 -11223.771,E2 -11223.771} C_VEL
LIN {X 0,Y 397.521,Z 322.145,A -85,B 0,C 180,E1 -11224.005,E2 -11224.005} C_VEL
LIN {X 0,Y 402.392,Z 340.665,A -85,B 0,C 180,E1 -11224.901,E2 -11224.901} C_VEL
LIN {X 0,Y 405.865,Z 356.557,A -85,B 0,C 180,E1 -11225.83,E2 -11225.83} C_VEL
LIN {X 0,Y 406.991,Z 362.731,A -85,B 0,C 180,E1 -11226.236,E2 -11226.236} C_VEL
LIN {X 0,Y 405.839,Z 376.489,A -85,B 0,C 180,E1 -11227.068,E2 -11227.068} C_VEL
LIN {X 0,Y 404.359,Z 389.801,A -85,B 0,C 180,E1 -11228.057,E2 -11228.057} C_VEL
LIN {X 0,Y 402.843,Z 403.493,A -85,B 0,C 180,E1 -11229.312,E2 -11229.312} C_VEL
LIN {X 0,Y 401.522,Z 414.937,A -85,B 0,C 180,E1 -11230.575,E2 -11230.575} C_VEL
LIN {X 0,Y 400.255,Z 426.564,A -85,B 0,C 180,E1 -11232.105,E2 -11232.105} C_VEL
LIN {X 0,Y 399.04,Z 436.394,A -85,B 0,C 180,E1 -11233.632,E2 -11233.632} C_VEL
LIN {X 0,Y 397.947,Z 446.063,A -85,B 0,C 180,E1 -11235.424,E2 -11235.424} C_VEL
LIN {X 0,Y 397.181,Z 454.149,A -85,B 0,C 180,E1 -11237.221,E2 -11237.221} C_VEL
LIN {X 0,Y 396.522,Z 461.697,A -85,B 0,C 180,E1 -11239.274,E2 -11239.274} C_VEL
LIN {X 0,Y 396.118,Z 467.693,A -85,B 0,C 180,E1 -11241.326,E2 -11241.326} C_VEL
LIN {X 0,Y 395.938,Z 471.241,A -85,B 0,C 180,E1 -11242.862,E2 -11242.862} C_VEL
LIN {X 0,Y 395.823,Z 474.841,A -85,B 0,C 180,E1 -11244.907,E2 -11244.907} C_VEL
LIN {X 0,Y 395.771,Z 477.193,A -85,B 0,C 180,E1 -11246.946,E2 -11246.946} C_VEL
LIN {X 0,Y 395.846,Z 477.922,A -85,B 0,C 180,E1 -11247.965,E2 -11247.965} C_VEL
LIN {X 0,Y 395.741,Z 478.467,A -85,B 0,C 180,E1 -11250,E2 -11250} C_VEL
LIN {X 0,Y 395.848,Z 477.782,A -85,B 0,C 180,E1 -11252.035,E2 -11252.035} C_VEL
LIN {X 0,Y 395.755,Z 475.887,A -85,B 0,C 180,E1 -11254.073,E2 -11254.073} C_VEL
LIN {X 0,Y 395.93,Z 472.496,A -85,B 0,C 180,E1 -11256.264,E2 -11256.264} C_VEL
LIN {X 0,Y 396.054,Z 468.361,A -85,B 0,C 180,E1 -11258.161,E2 -11258.161} C_VEL
LIN {X 0,Y 396.351,Z 462.545,A -85,B 0,C 180,E1 -11260.214,E2 -11260.214} C_VEL
LIN {X 0,Y 396.984,Z 455.187,A -85,B 0,C 180,E1 -11262.266,E2 -11262.266} C_VEL
LIN {X 0,Y 397.656,Z 447.494,A -85,B 0,C 180,E1 -11264.038,E2 -11264.038} C_VEL
LIN {X 0,Y 398.631,Z 438.01,A -85,B 0,C 180,E1 -11265.859,E2 -11265.859} C_VEL
LIN {X 0,Y 399.877,Z 426.839,A -85,B 0,C 180,E1 -11267.649,E2 -11267.649} C_VEL
LIN {X 0,Y 401.211,Z 415.319,A -85,B 0,C 180,E1 -11269.199,E2 -11269.199} C_VEL
LIN {X 0,Y 402.73,Z 402.071,A -85,B 0,C 180,E1 -11270.694,E2 -11270.694} C_VEL
LIN {X 0,Y 404.321,Z 388.752,A -85,B 0,C 180,E1 -11271.945,E2 -11271.945} C_VEL
LIN {X 0,Y 405.96,Z 374.351,A -85,B 0,C 180,E1 -11273.06,E2 -11273.06} C_VEL
LIN {X 0,Y 407.094,Z 362.965,A -85,B 0,C 180,E1 -11273.797,E2 -11273.797} C_VEL
LIN {X 0,Y 404.302,Z 345.801,A -85,B 0,C 180,E1 -11275.03,E2 -11275.03} C_VEL
LIN {X 0,Y 401.755,Z 332.602,A -85,B 0,C 180,E1 -11275.88,E2 -11275.88} C_VEL
LIN {X 0,Y 398.319,Z 320.89,A -85,B 0,C 180,E1 -11276.683,E2 -11276.683} C_VEL
LIN {X 0,Y 397.366,Z 317.256,A -85,B 0,C 180,E1 -11276.94,E2 -11276.94} C_VEL
LIN {X 0,Y 397.891,Z 310.615,A -85,B 0,C 180,E1 -11280.061,E2 -11280.061} C_VEL
LIN {X 0,Y 398.578,Z 302.902,A -85,B 0,C 180,E1 -11284.031,E2 -11284.031} C_VEL
LIN {X 0,Y 399.341,Z 296.798,A -85,B 0,C 180,E1 -11287.632,E2 -11287.632} C_VEL
LIN {X 0,Y 399.989,Z 292.631,A -85,B 0,C 180,E1 -11290.55,E2 -11290.55} C_VEL
LIN {X 0,Y 400.285,Z 290.343,A -85,B 0,C 180,E1 -11292.489,E2 -11292.489} C_VEL
LIN {X 0,Y 400.139,Z 288.367,A -85,B 0,C 180,E1 -11294.633,E2 -11294.633} C_VEL
LIN {X 0,Y 399.834,Z 286.96,A -85,B 0,C 180,E1 -11296.724,E2 -11296.724} C_VEL
LIN {X 0,Y 399.242,Z 285.864,A -85,B 0,C 180,E1 -11299.359,E2 -11299.359} C_VEL
LIN {X 0,Y 398.622,Z 285.365,A -85,B 0,C 180,E1 -11302.503,E2 -11302.503} C_VEL
LIN {X 0,Y 398.042,Z 285.656,A -85,B 0,C 180,E1 -11306.084,E2 -11306.084} C_VEL
LIN {X 0,Y 397.643,Z 286.659,A -85,B 0,C 180,E1 -11309.577,E2 -11309.577} C_VEL
LIN {X 0,Y 398.873,Z 289.624,A -85,B 0,C 180,E1 -11309.848,E2 -11309.848} C_VEL
LIN {X 0,Y 401.555,Z 294.564,A -85,B 0,C 180,E1 -11310.369,E2 -11310.369} C_VEL
LIN {X 0,Y 405.852,Z 304.472,A -85,B 0,C 180,E1 -11311.317,E2 -11311.317} C_VEL
LIN {X 0,Y 408.438,Z 312.127,A -85,B 0,C 180,E1 -11311.999,E2 -11311.999} C_VEL
LIN {X 0,Y 408.449,Z 315.383,A -85,B 0,C 180,E1 -11312.199,E2 -11312.199} C_VEL
LIN {X 0,Y 406.989,Z 331.011,A -85,B 0,C 180,E1 -11313.195,E2 -11313.195} C_VEL
LIN {X 0,Y 405.535,Z 345.406,A -85,B 0,C 180,E1 -11314.326,E2 -11314.326} C_VEL
LIN {X 0,Y 404.078,Z 358.703,A -85,B 0,C 180,E1 -11315.602,E2 -11315.602} C_VEL
LIN {X 0,Y 402.668,Z 371.017,A -85,B 0,C 180,E1 -11317.013,E2 -11317.013} C_VEL
LIN {X 0,Y 401.377,Z 381.396,A -85,B 0,C 180,E1 -11318.426,E2 -11318.426} C_VEL
LIN {X 0,Y 400.087,Z 392.52,A -85,B 0,C 180,E1 -11320.236,E2 -11320.236} C_VEL
LIN {X 0,Y 398.914,Z 401.771,A -85,B 0,C 180,E1 -11322.058,E2 -11322.058} C_VEL
LIN {X 0,Y 397.934,Z 410.26,A -85,B 0,C 180,E1 -11324.113,E2 -11324.113} C_VEL
LIN {X 0,Y 397.218,Z 417.03,A -85,B 0,C 180,E1 -11326.181,E2 -11326.181} C_VEL
LIN {X 0,Y 396.693,Z 422.226,A -85,B 0,C 180,E1 -11328.245,E2 -11328.245} C_VEL
LIN {X 0,Y 396.369,Z 425.157,A -85,B 0,C 180,E1 -11329.787,E2 -11329.787} C_VEL
LIN {X 0,Y 396.137,Z 427.958,A -85,B 0,C 180,E1 -11331.841,E2 -11331.841} C_VEL
LIN {X 0,Y 396.088,Z 429.489,A -85,B 0,C 180,E1 -11333.889,E2 -11333.889} C_VEL
LIN {X 0,Y 395.967,Z 429.807,A -85,B 0,C 180,E1 -11335.929,E2 -11335.929} C_VEL
LIN {X 0,Y 395.998,Z 428.902,A -85,B 0,C 180,E1 -11337.966,E2 -11337.966} C_VEL
LIN {X 0,Y 395.952,Z 426.761,A -85,B 0,C 180,E1 -11340,E2 -11340} C_VEL
LIN {X 0,Y 396.111,Z 423.353,A -85,B 0,C 180,E1 -11342.034,E2 -11342.034} C_VEL
LIN {X 0,Y 396.562,Z 418.621,A -85,B 0,C 180,E1 -11344.065,E2 -11344.065} C_VEL
LIN {X 0,Y 396.881,Z 412.489,A -85,B 0,C 180,E1 -11346.099,E2 -11346.099} C_VEL
LIN {X 0,Y 397.478,Z 404.767,A -85,B 0,C 180,E1 -11348.132,E2 -11348.132} C_VEL
LIN {X 0,Y 398.211,Z 396.501,A -85,B 0,C 180,E1 -11349.909,E2 -11349.909} C_VEL
LIN {X 0,Y 399.201,Z 386.601,A -85,B 0,C 180,E1 -11351.681,E2 -11351.681} C_VEL
LIN {X 0,Y 400.09,Z 376.52,A -85,B 0,C 180,E1 -11353.201,E2 -11353.201} C_VEL
LIN {X 0,Y 401.282,Z 364.593,A -85,B 0,C 180,E1 -11354.712,E2 -11354.712} C_VEL
LIN {X 0,Y 402.449,Z 351.585,A -85,B 0,C 180,E1 -11356.089,E2 -11356.089} C_VEL
LIN {X 0,Y 403.537,Z 338.704,A -85,B 0,C 180,E1 -11357.222,E2 -11357.222} C_VEL
LIN {X 0,Y 404.577,Z 324.907,A -85,B 0,C 180,E1 -11358.221,E2 -11358.221} C_VEL
LIN {X 0,Y 405.557,Z 309.304,A -85,B 0,C 180,E1 -11359.122,E2 -11359.122} C_VEL
LIN {X 0,Y 401.206,Z 293.347,A -85,B 0,C 180,E1 -11360.087,E2 -11360.087} C_VEL
LIN {X 0,Y 396.227,Z 276.934,A -85,B 0,C 180,E1 -11360.914,E2 -11360.914} C_VEL
LIN {X 0,Y 396.305,Z 273.939,A -85,B 0,C 180,E1 -11364.072,E2 -11364.072} C_VEL
LIN {X 0,Y 396.339,Z 270.767,A -85,B 0,C 180,E1 -11367.548,E2 -11367.548} C_VEL
LIN {X 0,Y 396.727,Z 270.694,A -85,B 0,C 180,E1 -11370.913,E2 -11370.913} C_VEL
LIN {X 0,Y 396.998,Z 270.658,A -85,B 0,C 180,E1 -11374.506,E2 -11374.506} C_VEL
LIN {X 0,Y 397.094,Z 270.648,A -85,B 0,C 180,E1 -11377.208,E2 -11377.208} C_VEL
LIN {X 0,Y 397.104,Z 270.645,A -85,B 0,C 180,E1 -11380.445,E2 -11380.445} C_VEL
LIN {X 0,Y 397.103,Z 270.643,A -85,B 0,C 180,E1 -11383.649,E2 -11383.649} C_VEL
LIN {X 0,Y 397.105,Z 270.646,A -85,B 0,C 180,E1 -11386.521,E2 -11386.521} C_VEL
LIN {X 0,Y 397.116,Z 270.643,A -85,B 0,C 180,E1 -11390.423,E2 -11390.423} C_VEL
LIN {X 0,Y 397.111,Z 270.645,A -85,B 0,C 180,E1 -11394.265,E2 -11394.265} C_VEL
LIN {X 0,Y 397.118,Z 270.646,A -85,B 0,C 180,E1 -11396.727,E2 -11396.727} C_VEL
LIN {X 0,Y 397.128,Z 270.644,A -85,B 0,C 180,E1 -11400.296,E2 -11400.296} C_VEL
LIN {X 0,Y 397.197,Z 270.636,A -85,B 0,C 180,E1 -11402.61,E2 -11402.61} C_VEL
LIN {X 0,Y 397.128,Z 270.642,A -85,B 0,C 180,E1 -11405.981,E2 -11405.981} C_VEL
LIN {X 0,Y 397.142,Z 270.639,A -85,B 0,C 180,E1 -11409.705,E2 -11409.705} C_VEL
LIN {X 0,Y 397.185,Z 270.635,A -85,B 0,C 180,E1 -11412.845,E2 -11412.845} C_VEL
LIN {X 0,Y 397.232,Z 270.629,A -85,B 0,C 180,E1 -11416.703,E2 -11416.703} C_VEL
LIN {X 0,Y 397.22,Z 270.631,A -85,B 0,C 180,E1 -11419.809,E2 -11419.809} C_VEL
LIN {X 0,Y 397.297,Z 270.62,A -85,B 0,C 180,E1 -11422.887,E2 -11422.887} C_VEL
LIN {X 0,Y 397.241,Z 270.625,A -85,B 0,C 180,E1 -11424.925,E2 -11424.925} C_VEL
LIN {X 0,Y 397.45,Z 270.604,A -85,B 0,C 180,E1 -11427.973,E2 -11427.973} C_VEL
LIN {X 0,Y 397.578,Z 270.588,A -85,B 0,C 180,E1 -11430,E2 -11430} C_VEL
LIN {X 0,Y 397.371,Z 270.61,A -85,B 0,C 180,E1 -11433.042,E2 -11433.042} C_VEL
LIN {X 0,Y 397.349,Z 270.617,A -85,B 0,C 180,E1 -11436.092,E2 -11436.092} C_VEL
LIN {X 0,Y 397.239,Z 270.627,A -85,B 0,C 180,E1 -11439.162,E2 -11439.162} C_VEL
LIN {X 0,Y 397.222,Z 270.631,A -85,B 0,C 180,E1 -11442.258,E2 -11442.258} C_VEL
LIN {X 0,Y 397.182,Z 270.636,A -85,B 0,C 180,E1 -11445.392,E2 -11445.392} C_VEL
LIN {X 0,Y 397.161,Z 270.637,A -85,B 0,C 180,E1 -11448.574,E2 -11448.574} C_VEL
LIN {X 0,Y 397.122,Z 270.641,A -85,B 0,C 180,E1 -11450.5,E2 -11450.5} C_VEL
LIN {X 0,Y 396.412,Z 270.733,A -85,B 0,C 180,E1 -11451.346,E2 -11451.346} C_VEL
LIN {X 0,Y 393.548,Z 271.086,A -85,B 0,C 180,E1 -11452.723,E2 -11452.723} C_VEL
LIN {X 0,Y 391.161,Z 271.386,A -85,B 0,C 180,E1 -11453.836,E2 -11453.836} C_VEL
LIN {X 0,Y 390.153,Z 271.51,A -85,B 0,C 180,E1 -11454.696,E2 -11454.696} C_VEL
LIN {X 0,Y 390.079,Z 271.518,A -85,B 0,C 180,E1 -11454.987,E2 -11454.987} C_VEL
LIN {X 0,Y 390.1,Z 271.516,A -85,B 0,C 180,E1 -11458.02,E2 -11458.02} C_VEL
LIN {X 0,Y 390.027,Z 271.528,A -85,B 0,C 180,E1 -11461.504,E2 -11461.504} C_VEL
LIN {X 0,Y 390.088,Z 271.522,A -85,B 0,C 180,E1 -11465.207,E2 -11465.207} C_VEL
LIN {X 0,Y 390.062,Z 271.524,A -85,B 0,C 180,E1 -11469.096,E2 -11469.096} C_VEL
LIN {X 0,Y 390.033,Z 271.524,A -85,B 0,C 180,E1 -11472.372,E2 -11472.372} C_VEL
LIN {X 0,Y 390.047,Z 271.525,A -85,B 0,C 180,E1 -11475.354,E2 -11475.354} C_VEL
LIN {X 0,Y 390.035,Z 271.525,A -85,B 0,C 180,E1 -11478.187,E2 -11478.187} C_VEL
LIN {X 0,Y 390.094,Z 271.52,A -85,B 0,C 180,E1 -11480.908,E2 -11480.908} C_VEL
LIN {X 0,Y 390.088,Z 271.521,A -85,B 0,C 180,E1 -11484.793,E2 -11484.793} C_VEL
LIN {X 0,Y 390.028,Z 271.529,A -85,B 0,C 180,E1 -11488.496,E2 -11488.496} C_VEL
LIN {X 0,Y 390.121,Z 271.515,A -85,B 0,C 180,E1 -11492.07,E2 -11492.07} C_VEL
LIN {X 0,Y 390.079,Z 271.519,A -85,B 0,C 180,E1 -11495.519,E2 -11495.519} C_VEL
LIN {X 0,Y 390.092,Z 271.516,A -85,B 0,C 180,E1 -11499.53,E2 -11499.53} C_VEL
LIN {X 0,Y 390.142,Z 271.511,A -85,B 0,C 180,E1 -11503.248,E2 -11503.248} C_VEL
LIN {X 0,Y 390.199,Z 271.506,A -85,B 0,C 180,E1 -11506.561,E2 -11506.561} C_VEL
LIN {X 0,Y 390.172,Z 271.508,A -85,B 0,C 180,E1 -11509.623,E2 -11509.623} C_VEL
LIN {X 0,Y 390.251,Z 271.498,A -85,B 0,C 180,E1 -11512.758,E2 -11512.758} C_VEL
LIN {X 0,Y 390.213,Z 271.502,A -85,B 0,C 180,E1 -11514.833,E2 -11514.833} C_VEL
LIN {X 0,Y 390.421,Z 271.479,A -85,B 0,C 180,E1 -11517.937,E2 -11517.937} C_VEL
LIN {X 0,Y 390.546,Z 271.464,A -85,B 0,C 180,E1 -11520,E2 -11520} C_VEL
LIN {X 0,Y 390.314,Z 271.489,A -85,B 0,C 180,E1 -11523.096,E2 -11523.096} C_VEL
LIN {X 0,Y 390.292,Z 271.495,A -85,B 0,C 180,E1 -11526.202,E2 -11526.202} C_VEL
LIN {X 0,Y 390.196,Z 271.505,A -85,B 0,C 180,E1 -11529.329,E2 -11529.329} C_VEL
LIN {X 0,Y 390.174,Z 271.507,A -85,B 0,C 180,E1 -11532.483,E2 -11532.483} C_VEL
LIN {X 0,Y 390.142,Z 271.515,A -85,B 0,C 180,E1 -11535.676,E2 -11535.676} C_VEL
LIN {X 0,Y 390.108,Z 271.516,A -85,B 0,C 180,E1 -11538.922,E2 -11538.922} C_VEL
LIN {X 0,Y 390.05,Z 271.522,A -85,B 0,C 180,E1 -11542.233,E2 -11542.233} C_VEL
LIN {X 0,Y 390.062,Z 271.524,A -85,B 0,C 180,E1 -11545.621,E2 -11545.621} C_VEL
LIN {X 0,Y 390.032,Z 271.528,A -85,B 0,C 180,E1 -11549.111,E2 -11549.111} C_VEL
LIN {X 0,Y 390.045,Z 271.526,A -85,B 0,C 180,E1 -11552.721,E2 -11552.721} C_VEL
LIN {X 0,Y 390.103,Z 271.709,A -85,B 0,C 180,E1 -11555.735,E2 -11555.735} C_VEL
LIN {X 0,Y 390.914,Z 276.403,A -85,B 0,C 180,E1 -11558.994,E2 -11558.994} C_VEL
LIN {X 0,Y 391.969,Z 282.044,A -85,B 0,C 180,E1 -11562.681,E2 -11562.681} C_VEL
LIN {X 0,Y 392.88,Z 287.045,A -85,B 0,C 180,E1 -11565.761,E2 -11565.761} C_VEL
LIN {X 0,Y 393.275,Z 290.766,A -85,B 0,C 180,E1 -11567.922,E2 -11567.922} C_VEL
LIN {X 0,Y 392.971,Z 295.067,A -85,B 0,C 180,E1 -11570.266,E2 -11570.266} C_VEL
LIN {X 0,Y 392.289,Z 301.769,A -85,B 0,C 180,E1 -11573.757,E2 -11573.757} C_VEL
LIN {X 0,Y 391.684,Z 307.871,A -85,B 0,C 180,E1 -11576.82,E2 -11576.82} C_VEL
LIN {X 0,Y 391.073,Z 315.193,A -85,B 0,C 180,E1 -11580.382,E2 -11580.382} C_VEL
LIN {X 0,Y 390.543,Z 321.885,A -85,B 0,C 180,E1 -11583.537,E2 -11583.537} C_VEL
LIN {X 0,Y 395.222,Z 339.634,A -85,B 0,C 180,E1 -11584.411,E2 -11584.411} C_VEL
LIN {X 0,Y 398.804,Z 355.823,A -85,B 0,C 180,E1 -11585.374,E2 -11585.374} C_VEL
LIN {X 0,Y 400.291,Z 363.857,A -85,B 0,C 180,E1 -11585.92,E2 -11585.92} C_VEL
LIN {X 0,Y 399.041,Z 378.036,A -85,B 0,C 180,E1 -11586.816,E2 -11586.816} C_VEL
LIN {X 0,Y 397.393,Z 392.191,A -85,B 0,C 180,E1 -11587.925,E2 -11587.925} C_VEL
LIN {X 0,Y 395.848,Z 405.389,A -85,B 0,C 180,E1 -11589.201,E2 -11589.201} C_VEL
LIN {X 0,Y 394.303,Z 418.15,A -85,B 0,C 180,E1 -11590.697,E2 -11590.697} C_VEL
LIN {X 0,Y 392.96,Z 429.527,A -85,B 0,C 180,E1 -11592.299,E2 -11592.299} C_VEL
LIN {X 0,Y 391.633,Z 440.275,A -85,B 0,C 180,E1 -11594.117,E2 -11594.117} C_VEL
LIN {X 0,Y 390.574,Z 449.484,A -85,B 0,C 180,E1 -11595.994,E2 -11595.994} C_VEL
LIN {X 0,Y 389.829,Z 457.691,A -85,B 0,C 180,E1 -11598.034,E2 -11598.034} C_VEL
LIN {X 0,Y 389.218,Z 464.451,A -85,B 0,C 180,E1 -11600.123,E2 -11600.123} C_VEL
LIN {X 0,Y 388.912,Z 469.747,A -85,B 0,C 180,E1 -11602.211,E2 -11602.211} C_VEL
LIN {X 0,Y 388.774,Z 472.93,A -85,B 0,C 180,E1 -11603.853,E2 -11603.853} C_VEL
LIN {X 0,Y 388.674,Z 475.765,A -85,B 0,C 180,E1 -11605.852,E2 -11605.852} C_VEL
LIN {X 0,Y 388.76,Z 477.522,A -85,B 0,C 180,E1 -11607.928,E2 -11607.928} C_VEL
LIN {X 0,Y 388.672,Z 478.063,A -85,B 0,C 180,E1 -11610,E2 -11610} C_VEL
LIN {X 0,Y 388.781,Z 477.371,A -85,B 0,C 180,E1 -11612.072,E2 -11612.072} C_VEL
LIN {X 0,Y 388.682,Z 475.467,A -85,B 0,C 180,E1 -11614.148,E2 -11614.148} C_VEL
LIN {X 0,Y 388.832,Z 472.344,A -85,B 0,C 180,E1 -11616.226,E2 -11616.226} C_VEL
LIN {X 0,Y 388.976,Z 467.917,A -85,B 0,C 180,E1 -11618.311,E2 -11618.311} C_VEL
LIN {X 0,Y 389.299,Z 462.099,A -85,B 0,C 180,E1 -11620.401,E2 -11620.401} C_VEL
LIN {X 0,Y 389.981,Z 454.745,A -85,B 0,C 180,E1 -11622.489,E2 -11622.489} C_VEL
LIN {X 0,Y 390.692,Z 446.942,A -85,B 0,C 180,E1 -11624.32,E2 -11624.32} C_VEL
LIN {X 0,Y 391.726,Z 437.615,A -85,B 0,C 180,E1 -11626.146,E2 -11626.146} C_VEL
LIN {X 0,Y 393.038,Z 426.513,A -85,B 0,C 180,E1 -11627.966,E2 -11627.966} C_VEL
LIN {X 0,Y 394.495,Z 414.338,A -85,B 0,C 180,E1 -11629.636,E2 -11629.636} C_VEL
LIN {X 0,Y 396.059,Z 401.995,A -85,B 0,C 180,E1 -11631.059,E2 -11631.059} C_VEL
LIN {X 0,Y 397.913,Z 387.407,A -85,B 0,C 180,E1 -11632.454,E2 -11632.454} C_VEL
LIN {X 0,Y 399.622,Z 373.295,A -85,B 0,C 180,E1 -11633.565,E2 -11633.565} C_VEL
LIN {X 0,Y 400.602,Z 364.126,A -85,B 0,C 180,E1 -11634.18,E2 -11634.18} C_VEL
LIN {X 0,Y 397.961,Z 346.822,A -85,B 0,C 180,E1 -11635.497,E2 -11635.497} C_VEL
LIN {X 0,Y 395.666,Z 334.409,A -85,B 0,C 180,E1 -11636.364,E2 -11636.364} C_VEL
LIN {X 0,Y 392.581,Z 323.676,A -85,B 0,C 180,E1 -11637.161,E2 -11637.161} C_VEL
LIN {X 0,Y 391.334,Z 319.931,A -85,B 0,C 180,E1 -11637.456,E2 -11637.456} C_VEL
LIN {X 0,Y 390.451,Z 316.393,A -85,B 0,C 180,E1 -11637.733,E2 -11637.733} C_VEL
LIN {X 0,Y 390.994,Z 310.092,A -85,B 0,C 180,E1 -11640.823,E2 -11640.823} C_VEL
LIN {X 0,Y 391.614,Z 303.517,A -85,B 0,C 180,E1 -11644.358,E2 -11644.358} C_VEL
LIN {X 0,Y 392.348,Z 298.308,A -85,B 0,C 180,E1 -11647.52,E2 -11647.52} C_VEL
LIN {X 0,Y 392.901,Z 294.67,A -85,B 0,C 180,E1 -11650.087,E2 -11650.087} C_VEL
LIN {X 0,Y 393.331,Z 291.552,A -85,B 0,C 180,E1 -11652.764,E2 -11652.764} C_VEL
LIN {X 0,Y 393.229,Z 290.108,A -85,B 0,C 180,E1 -11654.365,E2 -11654.365} C_VEL
LIN {X 0,Y 393.073,Z 289.056,A -85,B 0,C 180,E1 -11655.789,E2 -11655.789} C_VEL
LIN {X 0,Y 392.503,Z 287.665,A -85,B 0,C 180,E1 -11658.509,E2 -11658.509} C_VEL
LIN {X 0,Y 391.944,Z 286.98,A -85,B 0,C 180,E1 -11661.128,E2 -11661.128} C_VEL
LIN {X 0,Y 391.401,Z 286.827,A -85,B 0,C 180,E1 -11663.903,E2 -11663.903} C_VEL
LIN {X 0,Y 390.911,Z 287.317,A -85,B 0,C 180,E1 -11667.36,E2 -11667.36} C_VEL
LIN {X 0,Y 390.763,Z 287.882,A -85,B 0,C 180,E1 -11668.8,E2 -11668.8} C_VEL
LIN {X 0,Y 392.038,Z 290.753,A -85,B 0,C 180,E1 -11669.099,E2 -11669.099} C_VEL
LIN {X 0,Y 393.134,Z 292.561,A -85,B 0,C 180,E1 -11669.324,E2 -11669.324} C_VEL
LIN {X 0,Y 397.815,Z 301.932,A -85,B 0,C 180,E1 -11670.353,E2 -11670.353} C_VEL
LIN {X 0,Y 401.995,Z 313.228,A -85,B 0,C 180,E1 -11671.464,E2 -11671.464} C_VEL
LIN {X 0,Y 402.479,Z 315.07,A -85,B 0,C 180,E1 -11671.628,E2 -11671.628} C_VEL
LIN {X 0,Y 400.914,Z 330.713,A -85,B 0,C 180,E1 -11672.63,E2 -11672.63} C_VEL
LIN {X 0,Y 399.354,Z 345.049,A -85,B 0,C 180,E1 -11673.773,E2 -11673.773} C_VEL
LIN {X 0,Y 397.648,Z 359.532,A -85,B 0,C 180,E1 -11675.181,E2 -11675.181} C_VEL
LIN {X 0,Y 396.145,Z 371.698,A -85,B 0,C 180,E1 -11676.612,E2 -11676.612} C_VEL
LIN {X 0,Y 394.569,Z 383.782,A -85,B 0,C 180,E1 -11678.31,E2 -11678.31} C_VEL
LIN {X 0,Y 393.199,Z 394.547,A -85,B 0,C 180,E1 -11680.147,E2 -11680.147} C_VEL
LIN {X 0,Y 392.072,Z 402.689,A -85,B 0,C 180,E1 -11681.814,E2 -11681.814} C_VEL
LIN {X 0,Y 391.079,Z 410.808,A -85,B 0,C 180,E1 -11683.827,E2 -11683.827} C_VEL
LIN {X 0,Y 390.272,Z 417.553,A -85,B 0,C 180,E1 -11685.93,E2 -11685.93} C_VEL
LIN {X 0,Y 389.715,Z 422.762,A -85,B 0,C 180,E1 -11688.031,E2 -11688.031} C_VEL
LIN {X 0,Y 389.349,Z 425.688,A -85,B 0,C 180,E1 -11689.601,E2 -11689.601} C_VEL
LIN {X 0,Y 389.095,Z 428.47,A -85,B 0,C 180,E1 -11691.692,E2 -11691.692} C_VEL
LIN {X 0,Y 389.012,Z 429.999,A -85,B 0,C 180,E1 -11693.777,E2 -11693.777} C_VEL
LIN {X 0,Y 388.884,Z 430.309,A -85,B 0,C 180,E1 -11695.855,E2 -11695.855} C_VEL
LIN {X 0,Y 388.985,Z 429.995,A -85,B 0,C 180,E1 -11696.893,E2 -11696.893} C_VEL
LIN {X 0,Y 388.879,Z 428.463,A -85,B 0,C 180,E1 -11698.965,E2 -11698.965} C_VEL
LIN {X 0,Y 388.923,Z 425.674,A -85,B 0,C 180,E1 -11701.036,E2 -11701.036} C_VEL
LIN {X 0,Y 389.235,Z 421.593,A -85,B 0,C 180,E1 -11703.105,E2 -11703.105} C_VEL
LIN {X 0,Y 389.705,Z 416.148,A -85,B 0,C 180,E1 -11705.174,E2 -11705.174} C_VEL
LIN {X 0,Y 390.074,Z 409.225,A -85,B 0,C 180,E1 -11707.246,E2 -11707.246} C_VEL
LIN {X 0,Y 390.774,Z 401.754,A -85,B 0,C 180,E1 -11709.054,E2 -11709.054} C_VEL
LIN {X 0,Y 391.663,Z 392.789,A -85,B 0,C 180,E1 -11710.86,E2 -11710.86} C_VEL
LIN {X 0,Y 392.684,Z 382.048,A -85,B 0,C 180,E1 -11712.665,E2 -11712.665} C_VEL
LIN {X 0,Y 393.831,Z 371.06,A -85,B 0,C 180,E1 -11714.204,E2 -11714.204} C_VEL
LIN {X 0,Y 395.007,Z 358.658,A -85,B 0,C 180,E1 -11715.667,E2 -11715.667} C_VEL
LIN {X 0,Y 396.045,Z 346.275,A -85,B 0,C 180,E1 -11716.893,E2 -11716.893} C_VEL
LIN {X 0,Y 397.346,Z 332.289,A -85,B 0,C 180,E1 -11718.031,E2 -11718.031} C_VEL
LIN {X 0,Y 398.271,Z 318.509,A -85,B 0,C 180,E1 -11718.951,E2 -11718.951} C_VEL
LIN {X 0,Y 398.807,Z 311.237,A -85,B 0,C 180,E1 -11719.356,E2 -11719.356} C_VEL
LIN {X 0,Y 395.174,Z 297.28,A -85,B 0,C 180,E1 -11720.24,E2 -11720.24} C_VEL
LIN {X 0,Y 390.185,Z 281.056,A -85,B 0,C 180,E1 -11721.099,E2 -11721.099} C_VEL
LIN {X 0,Y 389.174,Z 277.345,A -85,B 0,C 180,E1 -11721.268,E2 -11721.268} C_VEL
LIN {X 0,Y 389.232,Z 274.263,A -85,B 0,C 180,E1 -11724.538,E2 -11724.538} C_VEL
LIN {X 0,Y 389.235,Z 272.182,A -85,B 0,C 180,E1 -11726.834,E2 -11726.834} C_VEL
LIN {X 0,Y 389.338,Z 271.615,A -85,B 0,C 180,E1 -11727.991,E2 -11727.991} C_VEL
LIN {X 0,Y 389.604,Z 271.579,A -85,B 0,C 180,E1 -11730.338,E2 -11730.338} C_VEL
LIN {X 0,Y 389.925,Z 271.538,A -85,B 0,C 180,E1 -11733.969,E2 -11733.969} C_VEL
LIN {X 0,Y 390.047,Z 271.523,A -85,B 0,C 180,E1 -11736.485,E2 -11736.485} C_VEL
LIN {X 0,Y 390.064,Z 271.523,A -85,B 0,C 180,E1 -11739.217,E2 -11739.217} C_VEL
LIN {X 0,Y 390.042,Z 271.524,A -85,B 0,C 180,E1 -11742.374,E2 -11742.374} C_VEL
LIN {X 0,Y 390.047,Z 271.525,A -85,B 0,C 180,E1 -11745.354,E2 -11745.354} C_VEL
LIN {X 0,Y 390.034,Z 271.525,A -85,B 0,C 180,E1 -11748.187,E2 -11748.187} C_VEL
LIN {X 0,Y 390.092,Z 271.521,A -85,B 0,C 180,E1 -11750.908,E2 -11750.908} C_VEL
LIN {X 0,Y 390.088,Z 271.521,A -85,B 0,C 180,E1 -11754.793,E2 -11754.793} C_VEL
LIN {X 0,Y 390.027,Z 271.529,A -85,B 0,C 180,E1 -11758.496,E2 -11758.496} C_VEL
LIN {X 0,Y 390.12,Z 271.515,A -85,B 0,C 180,E1 -11762.07,E2 -11762.07} C_VEL
LIN {X 0,Y 390.077,Z 271.518,A -85,B 0,C 180,E1 -11765.519,E2 -11765.519} C_VEL
LIN {X 0,Y 390.091,Z 271.517,A -85,B 0,C 180,E1 -11769.53,E2 -11769.53} C_VEL
LIN {X 0,Y 390.141,Z 271.511,A -85,B 0,C 180,E1 -11773.248,E2 -11773.248} C_VEL
LIN {X 0,Y 390.198,Z 271.507,A -85,B 0,C 180,E1 -11776.562,E2 -11776.562} C_VEL
LIN {X 0,Y 390.207,Z 271.505,A -85,B 0,C 180,E1 -11780.671,E2 -11780.671} C_VEL
LIN {X 0,Y 390.287,Z 271.495,A -85,B 0,C 180,E1 -11783.797,E2 -11783.797} C_VEL
LIN {X 0,Y 390.418,Z 271.48,A -85,B 0,C 180,E1 -11787.937,E2 -11787.937} C_VEL
LIN {X 0,Y 390.547,Z 271.464,A -85,B 0,C 180,E1 -11790,E2 -11790} C_VEL
LIN {X 0,Y 390.306,Z 271.49,A -85,B 0,C 180,E1 -11793.097,E2 -11793.097} C_VEL
LIN {X 0,Y 390.303,Z 271.493,A -85,B 0,C 180,E1 -11796.202,E2 -11796.202} C_VEL
LIN {X 0,Y 390.196,Z 271.505,A -85,B 0,C 180,E1 -11799.329,E2 -11799.329} C_VEL
LIN {X 0,Y 390.174,Z 271.507,A -85,B 0,C 180,E1 -11802.483,E2 -11802.483} C_VEL
LIN {X 0,Y 390.142,Z 271.515,A -85,B 0,C 180,E1 -11805.677,E2 -11805.677} C_VEL
LIN {X 0,Y 390.106,Z 271.516,A -85,B 0,C 180,E1 -11808.922,E2 -11808.922} C_VEL
LIN {X 0,Y 390.043,Z 271.522,A -85,B 0,C 180,E1 -11812.234,E2 -11812.234} C_VEL
LIN {X 0,Y 390.079,Z 271.518,A -85,B 0,C 180,E1 -11814.987,E2 -11814.987} C_VEL
LIN {X 0,Y 389.42,Z 271.603,A -85,B 0,C 180,E1 -11815.849,E2 -11815.849} C_VEL
LIN {X 0,Y 386.535,Z 271.963,A -85,B 0,C 180,E1 -11817.249,E2 -11817.249} C_VEL
LIN {X 0,Y 384.094,Z 272.263,A -85,B 0,C 180,E1 -11818.381,E2 -11818.381} C_VEL
LIN {X 0,Y 383.063,Z 272.397,A -85,B 0,C 180,E1 -11819.257,E2 -11819.257} C_VEL
LIN {X 0,Y 382.99,Z 272.402,A -85,B 0,C 180,E1 -11819.554,E2 -11819.554} C_VEL
LIN {X 0,Y 382.99,Z 272.402,A -85,B 0,C 180,E1 -11822.422,E2 -11822.422} C_VEL
LIN {X 0,Y 383.027,Z 272.396,A -85,B 0,C 180,E1 -11825.956,E2 -11825.956} C_VEL
LIN {X 0,Y 382.989,Z 272.404,A -85,B 0,C 180,E1 -11829.581,E2 -11829.581} C_VEL
LIN {X 0,Y 383.009,Z 272.402,A -85,B 0,C 180,E1 -11832.779,E2 -11832.779} C_VEL
LIN {X 0,Y 383,Z 272.401,A -85,B 0,C 180,E1 -11835.789,E2 -11835.789} C_VEL
LIN {X 0,Y 382.992,Z 272.405,A -85,B 0,C 180,E1 -11838.796,E2 -11838.796} C_VEL
LIN {X 0,Y 383.004,Z 272.4,A -85,B 0,C 180,E1 -11842.096,E2 -11842.096} C_VEL
LIN {X 0,Y 383.022,Z 272.398,A -85,B 0,C 180,E1 -11845.332,E2 -11845.332} C_VEL
LIN {X 0,Y 382.987,Z 272.404,A -85,B 0,C 180,E1 -11849.081,E2 -11849.081} C_VEL
LIN {X 0,Y 383.06,Z 272.397,A -85,B 0,C 180,E1 -11852.698,E2 -11852.698} C_VEL
LIN {X 0,Y 383.053,Z 272.395,A -85,B 0,C 180,E1 -11855.039,E2 -11855.039} C_VEL
LIN {X 0,Y 382.996,Z 272.404,A -85,B 0,C 180,E1 -11858.469,E2 -11858.469} C_VEL
LIN {X 0,Y 383.067,Z 272.393,A -85,B 0,C 180,E1 -11861.826,E2 -11861.826} C_VEL
LIN {X 0,Y 383.114,Z 272.386,A -85,B 0,C 180,E1 -11865.118,E2 -11865.118} C_VEL
LIN {X 0,Y 383.102,Z 272.391,A -85,B 0,C 180,E1 -11868.358,E2 -11868.358} C_VEL
LIN {X 0,Y 383.219,Z 272.376,A -85,B 0,C 180,E1 -11872.028,E2 -11872.028} C_VEL
LIN {X 0,Y 383.184,Z 272.378,A -85,B 0,C 180,E1 -11874.738,E2 -11874.738} C_VEL
LIN {X 0,Y 383.388,Z 272.355,A -85,B 0,C 180,E1 -11877.899,E2 -11877.899} C_VEL
LIN {X 0,Y 383.516,Z 272.34,A -85,B 0,C 180,E1 -11880,E2 -11880} C_VEL
LIN {X 0,Y 383.25,Z 272.369,A -85,B 0,C 180,E1 -11883.153,E2 -11883.153} C_VEL
LIN {X 0,Y 383.248,Z 272.371,A -85,B 0,C 180,E1 -11886.317,E2 -11886.317} C_VEL
LIN {X 0,Y 383.146,Z 272.385,A -85,B 0,C 180,E1 -11889.502,E2 -11889.502} C_VEL
LIN {X 0,Y 383.14,Z 272.383,A -85,B 0,C 180,E1 -11892.716,E2 -11892.716} C_VEL
LIN {X 0,Y 383.084,Z 272.392,A -85,B 0,C 180,E1 -11895.973,E2 -11895.973} C_VEL
LIN {X 0,Y 383.063,Z 272.395,A -85,B 0,C 180,E1 -11899.283,E2 -11899.283} C_VEL
LIN {X 0,Y 383.015,Z 272.398,A -85,B 0,C 180,E1 -11902.664,E2 -11902.664} C_VEL
LIN {X 0,Y 382.992,Z 272.405,A -85,B 0,C 180,E1 -11906.13,E2 -11906.13} C_VEL
LIN {X 0,Y 382.98,Z 272.405,A -85,B 0,C 180,E1 -11909.701,E2 -11909.701} C_VEL
LIN {X 0,Y 383.005,Z 272.403,A -85,B 0,C 180,E1 -11913.4,E2 -11913.4} C_VEL
LIN {X 0,Y 383.062,Z 272.42,A -85,B 0,C 180,E1 -11915.144,E2 -11915.144} C_VEL
LIN {X 0,Y 383.857,Z 277.146,A -85,B 0,C 180,E1 -11918.499,E2 -11918.499} C_VEL
LIN {X 0,Y 384.694,Z 281.602,A -85,B 0,C 180,E1 -11921.493,E2 -11921.493} C_VEL
LIN {X 0,Y 385.786,Z 287.573,A -85,B 0,C 180,E1 -11925.273,E2 -11925.273} C_VEL
LIN {X 0,Y 386.29,Z 291.631,A -85,B 0,C 180,E1 -11927.688,E2 -11927.688} C_VEL
LIN {X 0,Y 385.946,Z 296.536,A -85,B 0,C 180,E1 -11930.406,E2 -11930.406} C_VEL
LIN {X 0,Y 385.353,Z 302.115,A -85,B 0,C 180,E1 -11933.366,E2 -11933.366} C_VEL
LIN {X 0,Y 384.657,Z 308.745,A -85,B 0,C 180,E1 -11936.761,E2 -11936.761} C_VEL
LIN {X 0,Y 384.016,Z 316.07,A -85,B 0,C 180,E1 -11940.387,E2 -11940.387} C_VEL
LIN {X 0,Y 383.575,Z 321.58,A -85,B 0,C 180,E1 -11943.04,E2 -11943.04} C_VEL
LIN {X 0,Y 388.466,Z 340.384,A -85,B 0,C 180,E1 -11944.005,E2 -11944.005} C_VEL
LIN {X 0,Y 391.813,Z 355.398,A -85,B 0,C 180,E1 -11944.933,E2 -11944.933} C_VEL
LIN {X 0,Y 393.562,Z 364.999,A -85,B 0,C 180,E1 -11945.606,E2 -11945.606} C_VEL
LIN {X 0,Y 392.264,Z 379.226,A -85,B 0,C 180,E1 -11946.547,E2 -11946.547} C_VEL
LIN {X 0,Y 390.588,Z 392.917,A -85,B 0,C 180,E1 -11947.659,E2 -11947.659} C_VEL
LIN {X 0,Y 388.984,Z 405.918,A -85,B 0,C 180,E1 -11948.955,E2 -11948.955} C_VEL
LIN {X 0,Y 387.468,Z 417.919,A -85,B 0,C 180,E1 -11950.394,E2 -11950.394} C_VEL
LIN {X 0,Y 386.122,Z 428.968,A -85,B 0,C 180,E1 -11951.975,E2 -11951.975} C_VEL
LIN {X 0,Y 384.719,Z 439.739,A -85,B 0,C 180,E1 -11953.824,E2 -11953.824} C_VEL
LIN {X 0,Y 383.624,Z 448.746,A -85,B 0,C 180,E1 -11955.681,E2 -11955.681} C_VEL
LIN {X 0,Y 382.792,Z 457.201,A -85,B 0,C 180,E1 -11957.811,E2 -11957.811} C_VEL
LIN {X 0,Y 382.153,Z 463.986,A -85,B 0,C 180,E1 -11959.938,E2 -11959.938} C_VEL
LIN {X 0,Y 381.838,Z 469.305,A -85,B 0,C 180,E1 -11962.065,E2 -11962.065} C_VEL
LIN {X 0,Y 381.694,Z 472.719,A -85,B 0,C 180,E1 -11963.87,E2 -11963.87} C_VEL
LIN {X 0,Y 381.602,Z 475.346,A -85,B 0,C 180,E1 -11965.775,E2 -11965.775} C_VEL
LIN {X 0,Y 381.676,Z 477.112,A -85,B 0,C 180,E1 -11967.889,E2 -11967.889} C_VEL
LIN {X 0,Y 381.605,Z 477.653,A -85,B 0,C 180,E1 -11970,E2 -11970} C_VEL
LIN {X 0,Y 381.696,Z 476.958,A -85,B 0,C 180,E1 -11972.11,E2 -11972.11} C_VEL
LIN {X 0,Y 381.612,Z 475.052,A -85,B 0,C 180,E1 -11974.225,E2 -11974.225} C_VEL
LIN {X 0,Y 381.762,Z 471.927,A -85,B 0,C 180,E1 -11976.342,E2 -11976.342} C_VEL
LIN {X 0,Y 381.916,Z 467.499,A -85,B 0,C 180,E1 -11978.466,E2 -11978.466} C_VEL
LIN {X 0,Y 382.252,Z 461.684,A -85,B 0,C 180,E1 -11980.595,E2 -11980.595} C_VEL
LIN {X 0,Y 382.97,Z 454.348,A -85,B 0,C 180,E1 -11982.722,E2 -11982.722} C_VEL
LIN {X 0,Y 383.731,Z 446.57,A -85,B 0,C 180,E1 -11984.586,E2 -11984.586} C_VEL
LIN {X 0,Y 384.812,Z 437.282,A -85,B 0,C 180,E1 -11986.444,E2 -11986.444} C_VEL
LIN {X 0,Y 386.215,Z 426.279,A -85,B 0,C 180,E1 -11988.293,E2 -11988.293} C_VEL
LIN {X 0,Y 387.761,Z 414.227,A -85,B 0,C 180,E1 -11989.991,E2 -11989.991} C_VEL
LIN {X 0,Y 389.599,Z 400.814,A -85,B 0,C 180,E1 -11991.564,E2 -11991.564} C_VEL
LIN {X 0,Y 391.36,Z 387.739,A -85,B 0,C 180,E1 -11992.851,E2 -11992.851} C_VEL
LIN {X 0,Y 393.37,Z 372.272,A -85,B 0,C 180,E1 -11994.1,E2 -11994.1} C_VEL
LIN {X 0,Y 394.04,Z 364.714,A -85,B 0,C 180,E1 -11994.64,E2 -11994.64} C_VEL
LIN {X 0,Y 391.808,Z 348.771,A -85,B 0,C 180,E1 -11995.927,E2 -11995.927} C_VEL
LIN {X 0,Y 389.425,Z 335.193,A -85,B 0,C 180,E1 -11996.948,E2 -11996.948} C_VEL
LIN {X 0,Y 386.036,Z 323.564,A -85,B 0,C 180,E1 -11997.897,E2 -11997.897} C_VEL
LIN {X 0,Y 384.674,Z 319.525,A -85,B 0,C 180,E1 -11998.25,E2 -11998.25} C_VEL
LIN {X 0,Y 383.572,Z 315.948,A -85,B 0,C 180,E1 -11998.552,E2 -11998.552} C_VEL
LIN {X 0,Y 383.534,Z 315.535,A -85,B 0,C 180,E1 -11998.587,E2 -11998.587} C_VEL
LIN {X 0,Y 384.022,Z 309.972,A -85,B 0,C 180,E1 -12001.439,E2 -12001.439} C_VEL
LIN {X 0,Y 384.693,Z 304.135,A -85,B 0,C 180,E1 -12004.704,E2 -12004.704} C_VEL
LIN {X 0,Y 385.531,Z 298.516,A -85,B 0,C 180,E1 -12008.302,E2 -12008.302} C_VEL
LIN {X 0,Y 386.113,Z 295.051,A -85,B 0,C 180,E1 -12010.94,E2 -12010.94} C_VEL
LIN {X 0,Y 386.354,Z 292.538,A -85,B 0,C 180,E1 -12013.313,E2 -12013.313} C_VEL
LIN {X 0,Y 386.031,Z 290.322,A -85,B 0,C 180,E1 -12016.226,E2 -12016.226} C_VEL
LIN {X 0,Y 385.47,Z 289.026,A -85,B 0,C 180,E1 -12018.977,E2 -12018.977} C_VEL
LIN {X 0,Y 384.886,Z 288.389,A -85,B 0,C 180,E1 -12021.738,E2 -12021.738} C_VEL
LIN {X 0,Y 384.187,Z 288.398,A -85,B 0,C 180,E1 -12025.453,E2 -12025.453} C_VEL
LIN {X 0,Y 383.929,Z 289.017,A -85,B 0,C 180,E1 -12027.937,E2 -12027.937} C_VEL
LIN {X 0,Y 385.077,Z 291.737,A -85,B 0,C 180,E1 -12028.242,E2 -12028.242} C_VEL
LIN {X 0,Y 386.392,Z 293.782,A -85,B 0,C 180,E1 -12028.534,E2 -12028.534} C_VEL
LIN {X 0,Y 391.033,Z 302.552,A -85,B 0,C 180,E1 -12029.622,E2 -12029.622} C_VEL
LIN {X 0,Y 394.931,Z 312.44,A -85,B 0,C 180,E1 -12030.69,E2 -12030.69} C_VEL
LIN {X 0,Y 396.348,Z 316.984,A -85,B 0,C 180,E1 -12031.149,E2 -12031.149} C_VEL
LIN {X 0,Y 394.757,Z 332.174,A -85,B 0,C 180,E1 -12032.168,E2 -12032.168} C_VEL
LIN {X 0,Y 392.94,Z 347.465,A -85,B 0,C 180,E1 -12033.44,E2 -12033.44} C_VEL
LIN {X 0,Y 391.269,Z 360.473,A -85,B 0,C 180,E1 -12034.748,E2 -12034.748} C_VEL
LIN {X 0,Y 389.527,Z 373.537,A -85,B 0,C 180,E1 -12036.332,E2 -12036.332} C_VEL
LIN {X 0,Y 387.976,Z 384.493,A -85,B 0,C 180,E1 -12037.922,E2 -12037.922} C_VEL
LIN {X 0,Y 386.517,Z 395.203,A -85,B 0,C 180,E1 -12039.789,E2 -12039.789} C_VEL
LIN {X 0,Y 385.28,Z 403.57,A -85,B 0,C 180,E1 -12041.541,E2 -12041.541} C_VEL
LIN {X 0,Y 384.225,Z 411.386,A -85,B 0,C 180,E1 -12043.53,E2 -12043.53} C_VEL
LIN {X 0,Y 383.345,Z 418.134,A -85,B 0,C 180,E1 -12045.671,E2 -12045.671} C_VEL
LIN {X 0,Y 382.747,Z 423.304,A -85,B 0,C 180,E1 -12047.81,E2 -12047.81} C_VEL
LIN {X 0,Y 382.342,Z 426.227,A -85,B 0,C 180,E1 -12049.408,E2 -12049.408} C_VEL
LIN {X 0,Y 382.065,Z 429.007,A -85,B 0,C 180,E1 -12051.538,E2 -12051.538} C_VEL
LIN {X 0,Y 381.938,Z 430.518,A -85,B 0,C 180,E1 -12053.662,E2 -12053.662} C_VEL
LIN {X 0,Y 381.802,Z 430.81,A -85,B 0,C 180,E1 -12055.778,E2 -12055.778} C_VEL
LIN {X 0,Y 381.902,Z 430.489,A -85,B 0,C 180,E1 -12056.835,E2 -12056.835} C_VEL
LIN {X 0,Y 381.805,Z 428.936,A -85,B 0,C 180,E1 -12058.946,E2 -12058.946} C_VEL
LIN {X 0,Y 381.848,Z 426.12,A -85,B 0,C 180,E1 -12061.055,E2 -12061.055} C_VEL
LIN {X 0,Y 382.177,Z 422.006,A -85,B 0,C 180,E1 -12063.163,E2 -12063.163} C_VEL
LIN {X 0,Y 382.566,Z 418.031,A -85,B 0,C 180,E1 -12064.742,E2 -12064.742} C_VEL
LIN {X 0,Y 382.776,Z 413.243,A -85,B 0,C 180,E1 -12066.325,E2 -12066.325} C_VEL
LIN {X 0,Y 383.451,Z 405.446,A -85,B 0,C 180,E1 -12068.432,E2 -12068.432} C_VEL
LIN {X 0,Y 384.242,Z 397.105,A -85,B 0,C 180,E1 -12070.273,E2 -12070.273} C_VEL
LIN {X 0,Y 385.305,Z 387.123,A -85,B 0,C 180,E1 -12072.109,E2 -12072.109} C_VEL
LIN {X 0,Y 386.27,Z 376.958,A -85,B 0,C 180,E1 -12073.682,E2 -12073.682} C_VEL
LIN {X 0,Y 387.548,Z 364.945,A -85,B 0,C 180,E1 -12075.245,E2 -12075.245} C_VEL
LIN {X 0,Y 388.73,Z 352.338,A -85,B 0,C 180,E1 -12076.622,E2 -12076.622} C_VEL
LIN {X 0,Y 390.004,Z 338.886,A -85,B 0,C 180,E1 -12077.839,E2 -12077.839} C_VEL
LIN {X 0,Y 391.105,Z 325.009,A -85,B 0,C 180,E1 -12078.872,E2 -12078.872} C_VEL
LIN {X 0,Y 391.989,Z 313.148,A -85,B 0,C 180,E1 -12079.593,E2 -12079.593} C_VEL
LIN {X 0,Y 390.824,Z 307.344,A -85,B 0,C 180,E1 -12079.979,E2 -12079.979} C_VEL
LIN {X 0,Y 386.318,Z 291.621,A -85,B 0,C 180,E1 -12080.942,E2 -12080.942} C_VEL
LIN {X 0,Y 382.106,Z 277.702,A -85,B 0,C 180,E1 -12081.655,E2 -12081.655} C_VEL
LIN {X 0,Y 382.173,Z 274.568,A -85,B 0,C 180,E1 -12085.022,E2 -12085.022} C_VEL
LIN {X 0,Y 382.206,Z 272.506,A -85,B 0,C 180,E1 -12087.368,E2 -12087.368} C_VEL
LIN {X 0,Y 382.615,Z 272.452,A -85,B 0,C 180,E1 -12090.952,E2 -12090.952} C_VEL
LIN {X 0,Y 382.912,Z 272.413,A -85,B 0,C 180,E1 -12094.679,E2 -12094.679} C_VEL
LIN {X 0,Y 382.994,Z 272.404,A -85,B 0,C 180,E1 -12097.269,E2 -12097.269} C_VEL
LIN {X 0,Y 383.009,Z 272.399,A -85,B 0,C 180,E1 -12099.959,E2 -12099.959} C_VEL
LIN {X 0,Y 383.008,Z 272.402,A -85,B 0,C 180,E1 -12102.779,E2 -12102.779} C_VEL
LIN {X 0,Y 383,Z 272.4,A -85,B 0,C 180,E1 -12105.789,E2 -12105.789} C_VEL
LIN {X 0,Y 382.991,Z 272.405,A -85,B 0,C 180,E1 -12108.796,E2 -12108.796} C_VEL
LIN {X 0,Y 383.002,Z 272.4,A -85,B 0,C 180,E1 -12112.096,E2 -12112.096} C_VEL
LIN {X 0,Y 383.021,Z 272.398,A -85,B 0,C 180,E1 -12115.332,E2 -12115.332} C_VEL
LIN {X 0,Y 382.986,Z 272.404,A -85,B 0,C 180,E1 -12119.082,E2 -12119.082} C_VEL
LIN {X 0,Y 383.059,Z 272.397,A -85,B 0,C 180,E1 -12122.698,E2 -12122.698} C_VEL
LIN {X 0,Y 383.052,Z 272.395,A -85,B 0,C 180,E1 -12125.04,E2 -12125.04} C_VEL
LIN {X 0,Y 382.995,Z 272.404,A -85,B 0,C 180,E1 -12128.469,E2 -12128.469} C_VEL
LIN {X 0,Y 383.065,Z 272.392,A -85,B 0,C 180,E1 -12131.826,E2 -12131.826} C_VEL
LIN {X 0,Y 383.113,Z 272.387,A -85,B 0,C 180,E1 -12135.118,E2 -12135.118} C_VEL
LIN {X 0,Y 383.1,Z 272.391,A -85,B 0,C 180,E1 -12138.358,E2 -12138.358} C_VEL
LIN {X 0,Y 383.218,Z 272.376,A -85,B 0,C 180,E1 -12142.028,E2 -12142.028} C_VEL
LIN {X 0,Y 383.182,Z 272.377,A -85,B 0,C 180,E1 -12144.738,E2 -12144.738} C_VEL
LIN {X 0,Y 383.384,Z 272.356,A -85,B 0,C 180,E1 -12147.899,E2 -12147.899} C_VEL
LIN {X 0,Y 383.517,Z 272.34,A -85,B 0,C 180,E1 -12150,E2 -12150} C_VEL
LIN {X 0,Y 383.242,Z 272.37,A -85,B 0,C 180,E1 -12153.154,E2 -12153.154} C_VEL
LIN {X 0,Y 383.259,Z 272.37,A -85,B 0,C 180,E1 -12156.317,E2 -12156.317} C_VEL
LIN {X 0,Y 383.146,Z 272.385,A -85,B 0,C 180,E1 -12159.502,E2 -12159.502} C_VEL
LIN {X 0,Y 383.129,Z 272.387,A -85,B 0,C 180,E1 -12163.536,E2 -12163.536} C_VEL
LIN {X 0,Y 383.098,Z 272.392,A -85,B 0,C 180,E1 -12167.454,E2 -12167.454} C_VEL
LIN {X 0,Y 383.032,Z 272.396,A -85,B 0,C 180,E1 -12170.647,E2 -12170.647} C_VEL
LIN {X 0,Y 383.037,Z 272.398,A -85,B 0,C 180,E1 -12173.807,E2 -12173.807} C_VEL
LIN {X 0,Y 383.083,Z 272.391,A -85,B 0,C 180,E1 -12176.123,E2 -12176.123} C_VEL
LIN {X 0,Y 382.99,Z 272.402,A -85,B 0,C 180,E1 -12179.554,E2 -12179.554} C_VEL
LIN {X 0,Y 382.347,Z 272.487,A -85,B 0,C 180,E1 -12180.431,E2 -12180.431} C_VEL
LIN {X 0,Y 379.495,Z 272.843,A -85,B 0,C 180,E1 -12181.858,E2 -12181.858} C_VEL
LIN {X 0,Y 377.072,Z 273.142,A -85,B 0,C 180,E1 -12183.012,E2 -12183.012} C_VEL
LIN {X 0,Y 376.042,Z 273.268,A -85,B 0,C 180,E1 -12183.904,E2 -12183.904} C_VEL
LIN {X 0,Y 375.964,Z 273.276,A -85,B 0,C 180,E1 -12184.206,E2 -12184.206} C_VEL
LIN {X 0,Y 375.955,Z 273.279,A -85,B 0,C 180,E1 -12186.741,E2 -12186.741} C_VEL
LIN {X 0,Y 375.941,Z 273.28,A -85,B 0,C 180,E1 -12189.962,E2 -12189.962} C_VEL
LIN {X 0,Y 375.928,Z 273.281,A -85,B 0,C 180,E1 -12193.767,E2 -12193.767} C_VEL
LIN {X 0,Y 375.937,Z 273.283,A -85,B 0,C 180,E1 -12196.811,E2 -12196.811} C_VEL
LIN {X 0,Y 375.967,Z 273.278,A -85,B 0,C 180,E1 -12200.538,E2 -12200.538} C_VEL
LIN {X 0,Y 375.967,Z 273.277,A -85,B 0,C 180,E1 -12203.496,E2 -12203.496} C_VEL
LIN {X 0,Y 375.964,Z 273.276,A -85,B 0,C 180,E1 -12205.889,E2 -12205.889} C_VEL
LIN {X 0,Y 375.969,Z 273.276,A -85,B 0,C 180,E1 -12209.687,E2 -12209.687} C_VEL
LIN {X 0,Y 376.023,Z 273.268,A -85,B 0,C 180,E1 -12213.348,E2 -12213.348} C_VEL
LIN {X 0,Y 375.982,Z 273.277,A -85,B 0,C 180,E1 -12216.887,E2 -12216.887} C_VEL
LIN {X 0,Y 376.002,Z 273.276,A -85,B 0,C 180,E1 -12220.339,E2 -12220.339} C_VEL
LIN {X 0,Y 376.033,Z 273.269,A -85,B 0,C 180,E1 -12223.719,E2 -12223.719} C_VEL
LIN {X 0,Y 376.108,Z 273.258,A -85,B 0,C 180,E1 -12227.042,E2 -12227.042} C_VEL
LIN {X 0,Y 376.118,Z 273.261,A -85,B 0,C 180,E1 -12230.318,E2 -12230.318} C_VEL
LIN {X 0,Y 376.203,Z 273.247,A -85,B 0,C 180,E1 -12233.564,E2 -12233.564} C_VEL
LIN {X 0,Y 376.354,Z 273.232,A -85,B 0,C 180,E1 -12237.859,E2 -12237.859} C_VEL
LIN {X 0,Y 376.485,Z 273.216,A -85,B 0,C 180,E1 -12240,E2 -12240} C_VEL
LIN {X 0,Y 376.188,Z 273.249,A -85,B 0,C 180,E1 -12243.213,E2 -12243.213} C_VEL
LIN {X 0,Y 376.206,Z 273.247,A -85,B 0,C 180,E1 -12246.435,E2 -12246.435} C_VEL
LIN {X 0,Y 376.116,Z 273.262,A -85,B 0,C 180,E1 -12249.681,E2 -12249.681} C_VEL
LIN {X 0,Y 376.093,Z 273.264,A -85,B 0,C 180,E1 -12253.657,E2 -12253.657} C_VEL
LIN {X 0,Y 376.046,Z 273.27,A -85,B 0,C 180,E1 -12257.607,E2 -12257.607} C_VEL
LIN {X 0,Y 375.981,Z 273.274,A -85,B 0,C 180,E1 -12260.832,E2 -12260.832} C_VEL
LIN {X 0,Y 375.981,Z 273.275,A -85,B 0,C 180,E1 -12264.282,E2 -12264.282} C_VEL
LIN {X 0,Y 375.931,Z 273.282,A -85,B 0,C 180,E1 -12267.864,E2 -12267.864} C_VEL
LIN {X 0,Y 375.959,Z 273.281,A -85,B 0,C 180,E1 -12271.562,E2 -12271.562} C_VEL
LIN {X 0,Y 375.982,Z 273.317,A -85,B 0,C 180,E1 -12274.667,E2 -12274.667} C_VEL
LIN {X 0,Y 376.902,Z 278.535,A -85,B 0,C 180,E1 -12278.448,E2 -12278.448} C_VEL
LIN {X 0,Y 377.874,Z 283.818,A -85,B 0,C 180,E1 -12282.033,E2 -12282.033} C_VEL
LIN {X 0,Y 378.776,Z 288.705,A -85,B 0,C 180,E1 -12285.164,E2 -12285.164} C_VEL
LIN {X 0,Y 379.175,Z 291.219,A -85,B 0,C 180,E1 -12286.701,E2 -12286.701} C_VEL
LIN {X 0,Y 379.182,Z 294.928,A -85,B 0,C 180,E1 -12288.854,E2 -12288.854} C_VEL
LIN {X 0,Y 378.557,Z 301.054,A -85,B 0,C 180,E1 -12292.218,E2 -12292.218} C_VEL
LIN {X 0,Y 377.899,Z 307.242,A -85,B 0,C 180,E1 -12295.484,E2 -12295.484} C_VEL
LIN {X 0,Y 377.211,Z 314.103,A -85,B 0,C 180,E1 -12298.986,E2 -12298.986} C_VEL
LIN {X 0,Y 376.578,Z 321.297,A -85,B 0,C 180,E1 -12302.546,E2 -12302.546} C_VEL
LIN {X 0,Y 381.518,Z 340.287,A -85,B 0,C 180,E1 -12303.551,E2 -12303.551} C_VEL
LIN {X 0,Y 384.99,Z 355.739,A -85,B 0,C 180,E1 -12304.533,E2 -12304.533} C_VEL
LIN {X 0,Y 386.838,Z 366.28,A -85,B 0,C 180,E1 -12305.3,E2 -12305.3} C_VEL
LIN {X 0,Y 385.353,Z 381.287,A -85,B 0,C 180,E1 -12306.345,E2 -12306.345} C_VEL
LIN {X 0,Y 383.573,Z 394.903,A -85,B 0,C 180,E1 -12307.512,E2 -12307.512} C_VEL
LIN {X 0,Y 381.967,Z 407.492,A -85,B 0,C 180,E1 -12308.833,E2 -12308.833} C_VEL
LIN {X 0,Y 380.401,Z 419.357,A -85,B 0,C 180,E1 -12310.323,E2 -12310.323} C_VEL
LIN {X 0,Y 379.05,Z 429.949,A -85,B 0,C 180,E1 -12311.907,E2 -12311.907} C_VEL
LIN {X 0,Y 377.625,Z 440.5,A -85,B 0,C 180,E1 -12313.789,E2 -12313.789} C_VEL
LIN {X 0,Y 376.518,Z 449.316,A -85,B 0,C 180,E1 -12315.681,E2 -12315.681} C_VEL
LIN {X 0,Y 375.769,Z 456.682,A -85,B 0,C 180,E1 -12317.579,E2 -12317.579} C_VEL
LIN {X 0,Y 375.105,Z 463.5,A -85,B 0,C 180,E1 -12319.747,E2 -12319.747} C_VEL
LIN {X 0,Y 374.785,Z 468.845,A -85,B 0,C 180,E1 -12321.915,E2 -12321.915} C_VEL
LIN {X 0,Y 374.617,Z 472.483,A -85,B 0,C 180,E1 -12323.881,E2 -12323.881} C_VEL
LIN {X 0,Y 374.531,Z 474.916,A -85,B 0,C 180,E1 -12325.695,E2 -12325.695} C_VEL
LIN {X 0,Y 374.579,Z 476.693,A -85,B 0,C 180,E1 -12327.849,E2 -12327.849} C_VEL
LIN {X 0,Y 374.541,Z 477.237,A -85,B 0,C 180,E1 -12330,E2 -12330} C_VEL
LIN {X 0,Y 374.598,Z 476.546,A -85,B 0,C 180,E1 -12332.15,E2 -12332.15} C_VEL
LIN {X 0,Y 374.542,Z 474.643,A -85,B 0,C 180,E1 -12334.304,E2 -12334.304} C_VEL
LIN {X 0,Y 374.674,Z 471.522,A -85,B 0,C 180,E1 -12336.462,E2 -12336.462} C_VEL
LIN {X 0,Y 374.832,Z 467.104,A -85,B 0,C 180,E1 -12338.627,E2 -12338.627} C_VEL
LIN {X 0,Y 375.216,Z 461.302,A -85,B 0,C 180,E1 -12340.796,E2 -12340.796} C_VEL
LIN {X 0,Y 375.948,Z 453.993,A -85,B 0,C 180,E1 -12342.963,E2 -12342.963} C_VEL
LIN {X 0,Y 376.925,Z 444.996,A -85,B 0,C 180,E1 -12345.132,E2 -12345.132} C_VEL
LIN {X 0,Y 378.1,Z 435.553,A -85,B 0,C 180,E1 -12347.023,E2 -12347.023} C_VEL
LIN {X 0,Y 379.581,Z 424.734,A -85,B 0,C 180,E1 -12348.845,E2 -12348.845} C_VEL
LIN {X 0,Y 381.363,Z 412.035,A -85,B 0,C 180,E1 -12350.637,E2 -12350.637} C_VEL
LIN {X 0,Y 383.366,Z 398.575,A -85,B 0,C 180,E1 -12352.216,E2 -12352.216} C_VEL
LIN {X 0,Y 385.44,Z 383.868,A -85,B 0,C 180,E1 -12353.65,E2 -12353.65} C_VEL
LIN {X 0,Y 387.466,Z 368.988,A -85,B 0,C 180,E1 -12354.839,E2 -12354.839} C_VEL
LIN {X 0,Y 387.737,Z 366.762,A -85,B 0,C 180,E1 -12355.003,E2 -12355.003} C_VEL
LIN {X 0,Y 385.708,Z 350.702,A -85,B 0,C 180,E1 -12356.383,E2 -12356.383} C_VEL
LIN {X 0,Y 383.771,Z 338.62,A -85,B 0,C 180,E1 -12357.354,E2 -12357.354} C_VEL
LIN {X 0,Y 380.732,Z 327.112,A -85,B 0,C 180,E1 -12358.368,E2 -12358.368} C_VEL
LIN {X 0,Y 377.995,Z 318.973,A -85,B 0,C 180,E1 -12359.144,E2 -12359.144} C_VEL
LIN {X 0,Y 376.821,Z 315.669,A -85,B 0,C 180,E1 -12359.476,E2 -12359.476} C_VEL
LIN {X 0,Y 376.695,Z 314.575,A -85,B 0,C 180,E1 -12359.562,E2 -12359.562} C_VEL
LIN {X 0,Y 377.334,Z 308.162,A -85,B 0,C 180,E1 -12363.056,E2 -12363.056} C_VEL
LIN {X 0,Y 378.099,Z 302.517,A -85,B 0,C 180,E1 -12366.499,E2 -12366.499} C_VEL
LIN {X 0,Y 378.715,Z 298.786,A -85,B 0,C 180,E1 -12369.121,E2 -12369.121} C_VEL
LIN {X 0,Y 379.085,Z 296.999,A -85,B 0,C 180,E1 -12370.526,E2 -12370.526} C_VEL
LIN {X 0,Y 379.404,Z 294.088,A -85,B 0,C 180,E1 -12373.266,E2 -12373.266} C_VEL
LIN {X 0,Y 379.248,Z 292.503,A -85,B 0,C 180,E1 -12375.236,E2 -12375.236} C_VEL
LIN {X 0,Y 379.061,Z 291.581,A -85,B 0,C 180,E1 -12376.686,E2 -12376.686} C_VEL
LIN {X 0,Y 378.388,Z 290.36,A -85,B 0,C 180,E1 -12379.598,E2 -12379.598} C_VEL
LIN {X 0,Y 377.841,Z 289.845,A -85,B 0,C 180,E1 -12382.134,E2 -12382.134} C_VEL
LIN {X 0,Y 377.314,Z 289.806,A -85,B 0,C 180,E1 -12385.041,E2 -12385.041} C_VEL
LIN {X 0,Y 377.081,Z 290.155,A -85,B 0,C 180,E1 -12386.96,E2 -12386.96} C_VEL
LIN {X 0,Y 378.278,Z 292.915,A -85,B 0,C 180,E1 -12387.314,E2 -12387.314} C_VEL
LIN {X 0,Y 379.636,Z 294.857,A -85,B 0,C 180,E1 -12387.641,E2 -12387.641} C_VEL
LIN {X 0,Y 384.434,Z 303.749,A -85,B 0,C 180,E1 -12388.872,E2 -12388.872} C_VEL
LIN {X 0,Y 388.435,Z 313.183,A -85,B 0,C 180,E1 -12390.012,E2 -12390.012} C_VEL
LIN {X 0,Y 390.283,Z 319.084,A -85,B 0,C 180,E1 -12390.649,E2 -12390.649} C_VEL
LIN {X 0,Y 388.648,Z 333.765,A -85,B 0,C 180,E1 -12391.69,E2 -12391.69} C_VEL
LIN {X 0,Y 386.72,Z 348.8,A -85,B 0,C 180,E1 -12392.978,E2 -12392.978} C_VEL
LIN {X 0,Y 384.79,Z 362.73,A -85,B 0,C 180,E1 -12394.437,E2 -12394.437} C_VEL
LIN {X 0,Y 383.082,Z 374.464,A -85,B 0,C 180,E1 -12395.909,E2 -12395.909} C_VEL
LIN {X 0,Y 381.419,Z 385.298,A -85,B 0,C 180,E1 -12397.522,E2 -12397.522} C_VEL
LIN {X 0,Y 379.858,Z 395.929,A -85,B 0,C 180,E1 -12399.419,E2 -12399.419} C_VEL
LIN {X 0,Y 378.467,Z 404.558,A -85,B 0,C 180,E1 -12401.273,E2 -12401.273} C_VEL
LIN {X 0,Y 377.388,Z 412.03,A -85,B 0,C 180,E1 -12403.223,E2 -12403.223} C_VEL
LIN {X 0,Y 376.419,Z 418.724,A -85,B 0,C 180,E1 -12405.401,E2 -12405.401} C_VEL
LIN {X 0,Y 375.786,Z 423.891,A -85,B 0,C 180,E1 -12407.58,E2 -12407.58} C_VEL
LIN {X 0,Y 375.322,Z 426.795,A -85,B 0,C 180,E1 -12409.208,E2 -12409.208} C_VEL
LIN {X 0,Y 375.017,Z 429.543,A -85,B 0,C 180,E1 -12411.378,E2 -12411.378} C_VEL
LIN {X 0,Y 374.866,Z 431.044,A -85,B 0,C 180,E1 -12413.541,E2 -12413.541} C_VEL
LIN {X 0,Y 374.725,Z 431.314,A -85,B 0,C 180,E1 -12415.698,E2 -12415.698} C_VEL
LIN {X 0,Y 374.797,Z 430.346,A -85,B 0,C 180,E1 -12417.851,E2 -12417.851} C_VEL
LIN {X 0,Y 374.722,Z 428.142,A -85,B 0,C 180,E1 -12420,E2 -12420} C_VEL
LIN {X 0,Y 374.908,Z 424.658,A -85,B 0,C 180,E1 -12422.149,E2 -12422.149} C_VEL
LIN {X 0,Y 375.42,Z 419.832,A -85,B 0,C 180,E1 -12424.295,E2 -12424.295} C_VEL
LIN {X 0,Y 375.733,Z 413.595,A -85,B 0,C 180,E1 -12426.444,E2 -12426.444} C_VEL
LIN {X 0,Y 376.445,Z 405.751,A -85,B 0,C 180,E1 -12428.59,E2 -12428.59} C_VEL
LIN {X 0,Y 377.264,Z 397.36,A -85,B 0,C 180,E1 -12430.465,E2 -12430.465} C_VEL
LIN {X 0,Y 378.372,Z 387.323,A -85,B 0,C 180,E1 -12432.334,E2 -12432.334} C_VEL
LIN {X 0,Y 379.374,Z 377.102,A -85,B 0,C 180,E1 -12433.936,E2 -12433.936} C_VEL
LIN {X 0,Y 380.689,Z 365.027,A -85,B 0,C 180,E1 -12435.527,E2 -12435.527} C_VEL
LIN {X 0,Y 381.959,Z 351.91,A -85,B 0,C 180,E1 -12436.973,E2 -12436.973} C_VEL
LIN {X 0,Y 383.38,Z 337.278,A -85,B 0,C 180,E1 -12438.297,E2 -12438.297} C_VEL
LIN {X 0,Y 384.58,Z 322.106,A -85,B 0,C 180,E1 -12439.4,E2 -12439.4} C_VEL
LIN {X 0,Y 385.205,Z 314.245,A -85,B 0,C 180,E1 -12439.873,E2 -12439.873} C_VEL
LIN {X 0,Y 382.805,Z 304.274,A -85,B 0,C 180,E1 -12440.556,E2 -12440.556} C_VEL
LIN {X 0,Y 378.183,Z 288.432,A -85,B 0,C 180,E1 -12441.519,E2 -12441.519} C_VEL
LIN {X 0,Y 375.062,Z 278.063,A -85,B 0,C 180,E1 -12442.082,E2 -12442.082} C_VEL
LIN {X 0,Y 375.133,Z 274.873,A -85,B 0,C 180,E1 -12445.525,E2 -12445.525} C_VEL
LIN {X 0,Y 375.134,Z 273.808,A -85,B 0,C 180,E1 -12446.72,E2 -12446.72} C_VEL
LIN {X 0,Y 375.282,Z 273.366,A -85,B 0,C 180,E1 -12448.335,E2 -12448.335} C_VEL
LIN {X 0,Y 375.631,Z 273.322,A -85,B 0,C 180,E1 -12451.593,E2 -12451.593} C_VEL
LIN {X 0,Y 375.908,Z 273.286,A -85,B 0,C 180,E1 -12455.421,E2 -12455.421} C_VEL
LIN {X 0,Y 375.973,Z 273.275,A -85,B 0,C 180,E1 -12458.27,E2 -12458.27} C_VEL
LIN {X 0,Y 375.936,Z 273.281,A -85,B 0,C 180,E1 -12461.6,E2 -12461.6} C_VEL
LIN {X 0,Y 375.93,Z 273.283,A -85,B 0,C 180,E1 -12465.269,E2 -12465.269} C_VEL
LIN {X 0,Y 375.938,Z 273.282,A -85,B 0,C 180,E1 -12468.399,E2 -12468.399} C_VEL
LIN {X 0,Y 375.976,Z 273.275,A -85,B 0,C 180,E1 -12471.73,E2 -12471.73} C_VEL
LIN {X 0,Y 375.983,Z 273.275,A -85,B 0,C 180,E1 -12475.333,E2 -12475.333} C_VEL
LIN {X 0,Y 375.961,Z 273.28,A -85,B 0,C 180,E1 -12478.438,E2 -12478.438} C_VEL
LIN {X 0,Y 375.986,Z 273.276,A -85,B 0,C 180,E1 -12482.14,E2 -12482.14} C_VEL
LIN {X 0,Y 376.008,Z 273.276,A -85,B 0,C 180,E1 -12484.539,E2 -12484.539} C_VEL
LIN {X 0,Y 375.959,Z 273.28,A -85,B 0,C 180,E1 -12488.045,E2 -12488.045} C_VEL
LIN {X 0,Y 376.011,Z 273.27,A -85,B 0,C 180,E1 -12491.473,E2 -12491.473} C_VEL
LIN {X 0,Y 376.061,Z 273.266,A -85,B 0,C 180,E1 -12494.833,E2 -12494.833} C_VEL
LIN {X 0,Y 376.053,Z 273.27,A -85,B 0,C 180,E1 -12498.137,E2 -12498.137} C_VEL
LIN {X 0,Y 376.19,Z 273.252,A -85,B 0,C 180,E1 -12501.954,E2 -12501.954} C_VEL
LIN {X 0,Y 376.154,Z 273.253,A -85,B 0,C 180,E1 -12504.64,E2 -12504.64} C_VEL
LIN {X 0,Y 376.348,Z 273.233,A -85,B 0,C 180,E1 -12507.86,E2 -12507.86} C_VEL
LIN {X 0,Y 376.486,Z 273.216,A -85,B 0,C 180,E1 -12510,E2 -12510} C_VEL
LIN {X 0,Y 376.352,Z 273.231,A -85,B 0,C 180,E1 -12512.14,E2 -12512.14} C_VEL
LIN {X 0,Y 376.217,Z 273.246,A -85,B 0,C 180,E1 -12516.436,E2 -12516.436} C_VEL
LIN {X 0,Y 376.116,Z 273.262,A -85,B 0,C 180,E1 -12519.682,E2 -12519.682} C_VEL
LIN {X 0,Y 376.093,Z 273.264,A -85,B 0,C 180,E1 -12523.658,E2 -12523.658} C_VEL
LIN {X 0,Y 376.046,Z 273.27,A -85,B 0,C 180,E1 -12527.607,E2 -12527.607} C_VEL
LIN {X 0,Y 375.981,Z 273.275,A -85,B 0,C 180,E1 -12530.832,E2 -12530.832} C_VEL
LIN {X 0,Y 375.997,Z 273.272,A -85,B 0,C 180,E1 -12534.281,E2 -12534.281} C_VEL
LIN {X 0,Y 376.023,Z 273.27,A -85,B 0,C 180,E1 -12536.652,E2 -12536.652} C_VEL
LIN {X 0,Y 375.968,Z 273.276,A -85,B 0,C 180,E1 -12540.313,E2 -12540.313} C_VEL
LIN {X 0,Y 375.964,Z 273.276,A -85,B 0,C 180,E1 -12544.206,E2 -12544.206} C_VEL
LIN {X 0,Y 375.306,Z 273.362,A -85,B 0,C 180,E1 -12545.1,E2 -12545.1} C_VEL
LIN {X 0,Y 372.433,Z 273.716,A -85,B 0,C 180,E1 -12546.554,E2 -12546.554} C_VEL
LIN {X 0,Y 369.996,Z 274.021,A -85,B 0,C 180,E1 -12547.729,E2 -12547.729} C_VEL
LIN {X 0,Y 368.957,Z 274.151,A -85,B 0,C 180,E1 -12548.639,E2 -12548.639} C_VEL
LIN {X 0,Y 368.877,Z 274.163,A -85,B 0,C 180,E1 -12548.947,E2 -12548.947} C_VEL
LIN {X 0,Y 368.873,Z 274.159,A -85,B 0,C 180,E1 -12552.007,E2 -12552.007} C_VEL
LIN {X 0,Y 368.881,Z 274.162,A -85,B 0,C 180,E1 -12555.175,E2 -12555.175} C_VEL
LIN {X 0,Y 368.886,Z 274.158,A -85,B 0,C 180,E1 -12558.178,E2 -12558.178} C_VEL
LIN {X 0,Y 368.913,Z 274.156,A -85,B 0,C 180,E1 -12561.36,E2 -12561.36} C_VEL
LIN {X 0,Y 368.94,Z 274.153,A -85,B 0,C 180,E1 -12565.146,E2 -12565.146} C_VEL
LIN {X 0,Y 368.933,Z 274.155,A -85,B 0,C 180,E1 -12569.046,E2 -12569.046} C_VEL
LIN {X 0,Y 368.967,Z 274.151,A -85,B 0,C 180,E1 -12572.796,E2 -12572.796} C_VEL
LIN {X 0,Y 368.937,Z 274.154,A -85,B 0,C 180,E1 -12576.117,E2 -12576.117} C_VEL
LIN {X 0,Y 368.941,Z 274.152,A -85,B 0,C 180,E1 -12579.947,E2 -12579.947} C_VEL
LIN {X 0,Y 368.98,Z 274.146,A -85,B 0,C 180,E1 -12583.399,E2 -12583.399} C_VEL
LIN {X 0,Y 369.062,Z 274.137,A -85,B 0,C 180,E1 -12586.79,E2 -12586.79} C_VEL
LIN {X 0,Y 369.068,Z 274.14,A -85,B 0,C 180,E1 -12590.131,E2 -12590.131} C_VEL
LIN {X 0,Y 369.163,Z 274.124,A -85,B 0,C 180,E1 -12593.441,E2 -12593.441} C_VEL
LIN {X 0,Y 369.318,Z 274.108,A -85,B 0,C 180,E1 -12597.819,E2 -12597.819} C_VEL
LIN {X 0,Y 369.434,Z 274.094,A -85,B 0,C 180,E1 -12600,E2 -12600} C_VEL
LIN {X 0,Y 369.32,Z 274.107,A -85,B 0,C 180,E1 -12602.181,E2 -12602.181} C_VEL
LIN {X 0,Y 369.166,Z 274.123,A -85,B 0,C 180,E1 -12606.559,E2 -12606.559} C_VEL
LIN {X 0,Y 369.066,Z 274.139,A -85,B 0,C 180,E1 -12609.868,E2 -12609.868} C_VEL
LIN {X 0,Y 369.041,Z 274.144,A -85,B 0,C 180,E1 -12613.772,E2 -12613.772} C_VEL
LIN {X 0,Y 369.004,Z 274.147,A -85,B 0,C 180,E1 -12617.768,E2 -12617.768} C_VEL
LIN {X 0,Y 368.933,Z 274.155,A -85,B 0,C 180,E1 -12621.219,E2 -12621.219} C_VEL
LIN {X 0,Y 368.932,Z 274.153,A -85,B 0,C 180,E1 -12624.777,E2 -12624.777} C_VEL
LIN {X 0,Y 368.899,Z 274.158,A -85,B 0,C 180,E1 -12628.793,E2 -12628.793} C_VEL
LIN {X 0,Y 368.9,Z 274.16,A -85,B 0,C 180,E1 -12632.238,E2 -12632.238} C_VEL
LIN {X 0,Y 368.925,Z 274.192,A -85,B 0,C 180,E1 -12634.192,E2 -12634.192} C_VEL
LIN {X 0,Y 369.709,Z 278.607,A -85,B 0,C 180,E1 -12637.467,E2 -12637.467} C_VEL
LIN {X 0,Y 370.768,Z 284.49,A -85,B 0,C 180,E1 -12641.562,E2 -12641.562} C_VEL
LIN {X 0,Y 371.549,Z 288.839,A -85,B 0,C 180,E1 -12644.416,E2 -12644.416} C_VEL
LIN {X 0,Y 372.222,Z 293.26,A -85,B 0,C 180,E1 -12647.178,E2 -12647.178} C_VEL
LIN {X 0,Y 372.143,Z 296.492,A -85,B 0,C 180,E1 -12649.061,E2 -12649.061} C_VEL
LIN {X 0,Y 371.565,Z 301.87,A -85,B 0,C 180,E1 -12652.062,E2 -12652.062} C_VEL
LIN {X 0,Y 370.895,Z 307.986,A -85,B 0,C 180,E1 -12655.357,E2 -12655.357} C_VEL
LIN {X 0,Y 370.131,Z 315.297,A -85,B 0,C 180,E1 -12659.158,E2 -12659.158} C_VEL
LIN {X 0,Y 369.596,Z 321.035,A -85,B 0,C 180,E1 -12662.05,E2 -12662.05} C_VEL
LIN {X 0,Y 374.454,Z 339.887,A -85,B 0,C 180,E1 -12663.065,E2 -12663.065} C_VEL
LIN {X 0,Y 377.933,Z 355.191,A -85,B 0,C 180,E1 -12664.067,E2 -12664.067} C_VEL
LIN {X 0,Y 380.078,Z 367.165,A -85,B 0,C 180,E1 -12664.965,E2 -12664.965} C_VEL
LIN {X 0,Y 378.583,Z 382.02,A -85,B 0,C 180,E1 -12666.041,E2 -12666.041} C_VEL
LIN {X 0,Y 376.755,Z 395.41,A -85,B 0,C 180,E1 -12667.227,E2 -12667.227} C_VEL
LIN {X 0,Y 374.968,Z 408.989,A -85,B 0,C 180,E1 -12668.706,E2 -12668.706} C_VEL
LIN {X 0,Y 373.3,Z 420.925,A -85,B 0,C 180,E1 -12670.276,E2 -12670.276} C_VEL
LIN {X 0,Y 371.973,Z 430.887,A -85,B 0,C 180,E1 -12671.835,E2 -12671.835} C_VEL
LIN {X 0,Y 370.524,Z 441.224,A -85,B 0,C 180,E1 -12673.753,E2 -12673.753} C_VEL
LIN {X 0,Y 369.403,Z 449.852,A -85,B 0,C 180,E1 -12675.68,E2 -12675.68} C_VEL
LIN {X 0,Y 368.576,Z 457.965,A -85,B 0,C 180,E1 -12677.892,E2 -12677.892} C_VEL
LIN {X 0,Y 367.949,Z 464.43,A -85,B 0,C 180,E1 -12680.101,E2 -12680.101} C_VEL
LIN {X 0,Y 367.643,Z 469.444,A -85,B 0,C 180,E1 -12682.31,E2 -12682.31} C_VEL
LIN {X 0,Y 367.474,Z 473.114,A -85,B 0,C 180,E1 -12684.513,E2 -12684.513} C_VEL
LIN {X 0,Y 367.405,Z 475.518,A -85,B 0,C 180,E1 -12686.71,E2 -12686.71} C_VEL
LIN {X 0,Y 367.515,Z 476.704,A -85,B 0,C 180,E1 -12688.904,E2 -12688.904} C_VEL
LIN {X 0,Y 367.516,Z 476.628,A -85,B 0,C 180,E1 -12691.096,E2 -12691.096} C_VEL
LIN {X 0,Y 367.418,Z 475.338,A -85,B 0,C 180,E1 -12693.29,E2 -12693.29} C_VEL
LIN {X 0,Y 367.506,Z 472.841,A -85,B 0,C 180,E1 -12695.487,E2 -12695.487} C_VEL
LIN {X 0,Y 367.657,Z 469.097,A -85,B 0,C 180,E1 -12697.69,E2 -12697.69} C_VEL
LIN {X 0,Y 367.947,Z 464.021,A -85,B 0,C 180,E1 -12699.899,E2 -12699.899} C_VEL
LIN {X 0,Y 368.573,Z 457.519,A -85,B 0,C 180,E1 -12702.108,E2 -12702.108} C_VEL
LIN {X 0,Y 369.415,Z 449.432,A -85,B 0,C 180,E1 -12704.319,E2 -12704.319} C_VEL
LIN {X 0,Y 370.671,Z 439.576,A -85,B 0,C 180,E1 -12706.523,E2 -12706.523} C_VEL
LIN {X 0,Y 372.167,Z 429.276,A -85,B 0,C 180,E1 -12708.44,E2 -12708.44} C_VEL
LIN {X 0,Y 373.682,Z 418.97,A -85,B 0,C 180,E1 -12710.074,E2 -12710.074} C_VEL
LIN {X 0,Y 375.535,Z 406.956,A -85,B 0,C 180,E1 -12711.692,E2 -12711.692} C_VEL
LIN {X 0,Y 377.763,Z 392.759,A -85,B 0,C 180,E1 -12713.287,E2 -12713.287} C_VEL
LIN {X 0,Y 379.808,Z 379.29,A -85,B 0,C 180,E1 -12714.552,E2 -12714.552} C_VEL
LIN {X 0,Y 381.34,Z 368.201,A -85,B 0,C 180,E1 -12715.438,E2 -12715.438} C_VEL
LIN {X 0,Y 379.546,Z 351.608,A -85,B 0,C 180,E1 -12716.946,E2 -12716.946} C_VEL
LIN {X 0,Y 377.825,Z 340.32,A -85,B 0,C 180,E1 -12717.925,E2 -12717.925} C_VEL
LIN {X 0,Y 374.51,Z 327.369,A -85,B 0,C 180,E1 -12719.165,E2 -12719.165} C_VEL
LIN {X 0,Y 371.306,Z 318.127,A -85,B 0,C 180,E1 -12720.165,E2 -12720.165} C_VEL
LIN {X 0,Y 369.991,Z 314.557,A -85,B 0,C 180,E1 -12720.58,E2 -12720.58} C_VEL
LIN {X 0,Y 369.865,Z 313.486,A -85,B 0,C 180,E1 -12720.694,E2 -12720.694} C_VEL
LIN {X 0,Y 370.515,Z 307.717,A -85,B 0,C 180,E1 -12724.025,E2 -12724.025} C_VEL
LIN {X 0,Y 371.298,Z 302.6,A -85,B 0,C 180,E1 -12727.347,E2 -12727.347} C_VEL
LIN {X 0,Y 371.931,Z 299.119,A -85,B 0,C 180,E1 -12729.976,E2 -12729.976} C_VEL
LIN {X 0,Y 372.395,Z 296.221,A -85,B 0,C 180,E1 -12732.606,E2 -12732.606} C_VEL
LIN {X 0,Y 372.42,Z 294.737,A -85,B 0,C 180,E1 -12734.286,E2 -12734.286} C_VEL
LIN {X 0,Y 371.994,Z 292.88,A -85,B 0,C 180,E1 -12737.146,E2 -12737.146} C_VEL
LIN {X 0,Y 371.367,Z 291.788,A -85,B 0,C 180,E1 -12739.952,E2 -12739.952} C_VEL
LIN {X 0,Y 370.765,Z 291.295,A -85,B 0,C 180,E1 -12742.762,E2 -12742.762} C_VEL
LIN {X 0,Y 370.244,Z 291.434,A -85,B 0,C 180,E1 -12745.849,E2 -12745.849} C_VEL
LIN {X 0,Y 371.447,Z 294.197,A -85,B 0,C 180,E1 -12746.263,E2 -12746.263} C_VEL
LIN {X 0,Y 372.908,Z 295.986,A -85,B 0,C 180,E1 -12746.637,E2 -12746.637} C_VEL
LIN {X 0,Y 378.801,Z 306.808,A -85,B 0,C 180,E1 -12748.31,E2 -12748.31} C_VEL
LIN {X 0,Y 382.391,Z 315.255,A -85,B 0,C 180,E1 -12749.423,E2 -12749.423} C_VEL
LIN {X 0,Y 384.252,Z 321.203,A -85,B 0,C 180,E1 -12750.117,E2 -12750.117} C_VEL
LIN {X 0,Y 384.091,Z 324.813,A -85,B 0,C 180,E1 -12750.394,E2 -12750.394} C_VEL
LIN {X 0,Y 382.019,Z 340.172,A -85,B 0,C 180,E1 -12751.574,E2 -12751.574} C_VEL
LIN {X 0,Y 379.861,Z 354.915,A -85,B 0,C 180,E1 -12752.979,E2 -12752.979} C_VEL
LIN {X 0,Y 377.996,Z 367.256,A -85,B 0,C 180,E1 -12754.388,E2 -12754.388} C_VEL
LIN {X 0,Y 375.94,Z 379.862,A -85,B 0,C 180,E1 -12756.109,E2 -12756.109} C_VEL
LIN {X 0,Y 374.391,Z 389.379,A -85,B 0,C 180,E1 -12757.659,E2 -12757.659} C_VEL
LIN {X 0,Y 372.747,Z 399.358,A -85,B 0,C 180,E1 -12759.586,E2 -12759.586} C_VEL
LIN {X 0,Y 371.362,Z 407.644,A -85,B 0,C 180,E1 -12761.519,E2 -12761.519} C_VEL
LIN {X 0,Y 370.282,Z 414.483,A -85,B 0,C 180,E1 -12763.459,E2 -12763.459} C_VEL
LIN {X 0,Y 369.329,Z 420.753,A -85,B 0,C 180,E1 -12765.678,E2 -12765.678} C_VEL
LIN {X 0,Y 368.626,Z 425.508,A -85,B 0,C 180,E1 -12767.894,E2 -12767.894} C_VEL
LIN {X 0,Y 368.138,Z 428.904,A -85,B 0,C 180,E1 -12770.107,E2 -12770.107} C_VEL
LIN {X 0,Y 367.879,Z 430.996,A -85,B 0,C 180,E1 -12772.315,E2 -12772.315} C_VEL
LIN {X 0,Y 367.762,Z 431.844,A -85,B 0,C 180,E1 -12774.517,E2 -12774.517} C_VEL
LIN {X 0,Y 367.727,Z 431.47,A -85,B 0,C 180,E1 -12776.713,E2 -12776.713} C_VEL
LIN {X 0,Y 367.664,Z 429.863,A -85,B 0,C 180,E1 -12778.905,E2 -12778.905} C_VEL
LIN {X 0,Y 367.706,Z 426.987,A -85,B 0,C 180,E1 -12781.095,E2 -12781.095} C_VEL
LIN {X 0,Y 368.068,Z 422.802,A -85,B 0,C 180,E1 -12783.284,E2 -12783.284} C_VEL
LIN {X 0,Y 368.473,Z 418.76,A -85,B 0,C 180,E1 -12784.924,E2 -12784.924} C_VEL
LIN {X 0,Y 368.851,Z 412.094,A -85,B 0,C 180,E1 -12787.115,E2 -12787.115} C_VEL
LIN {X 0,Y 369.644,Z 403.751,A -85,B 0,C 180,E1 -12789.301,E2 -12789.301} C_VEL
LIN {X 0,Y 370.625,Z 394.881,A -85,B 0,C 180,E1 -12791.208,E2 -12791.208} C_VEL
LIN {X 0,Y 371.754,Z 384.254,A -85,B 0,C 180,E1 -12793.113,E2 -12793.113} C_VEL
LIN {X 0,Y 372.946,Z 373.412,A -85,B 0,C 180,E1 -12794.738,E2 -12794.738} C_VEL
LIN {X 0,Y 374.329,Z 360.522,A -85,B 0,C 180,E1 -12796.357,E2 -12796.357} C_VEL
LIN {X 0,Y 375.555,Z 347.687,A -85,B 0,C 180,E1 -12797.704,E2 -12797.704} C_VEL
LIN {X 0,Y 376.963,Z 333.801,A -85,B 0,C 180,E1 -12798.901,E2 -12798.901} C_VEL
LIN {X 0,Y 378.036,Z 319.569,A -85,B 0,C 180,E1 -12799.908,E2 -12799.908} C_VEL
LIN {X 0,Y 378.446,Z 315.387,A -85,B 0,C 180,E1 -12800.161,E2 -12800.161} C_VEL
LIN {X 0,Y 374.768,Z 301.011,A -85,B 0,C 180,E1 -12801.169,E2 -12801.169} C_VEL
LIN {X 0,Y 370.011,Z 285.175,A -85,B 0,C 180,E1 -12802.104,E2 -12802.104} C_VEL
LIN {X 0,Y 368.026,Z 278.45,A -85,B 0,C 180,E1 -12802.454,E2 -12802.454} C_VEL
LIN {X 0,Y 368.076,Z 275.059,A -85,B 0,C 180,E1 -12806.179,E2 -12806.179} C_VEL
LIN {X 0,Y 368.101,Z 274.263,A -85,B 0,C 180,E1 -12807.273,E2 -12807.273} C_VEL
LIN {X 0,Y 368.53,Z 274.206,A -85,B 0,C 180,E1 -12810.991,E2 -12810.991} C_VEL
LIN {X 0,Y 368.728,Z 274.18,A -85,B 0,C 180,E1 -12813.556,E2 -12813.556} C_VEL
LIN {X 0,Y 368.9,Z 274.156,A -85,B 0,C 180,E1 -12816.199,E2 -12816.199} C_VEL
LIN {X 0,Y 368.902,Z 274.161,A -85,B 0,C 180,E1 -12818.954,E2 -12818.954} C_VEL
LIN {X 0,Y 368.883,Z 274.158,A -85,B 0,C 180,E1 -12822.009,E2 -12822.009} C_VEL
LIN {X 0,Y 368.883,Z 274.162,A -85,B 0,C 180,E1 -12825.176,E2 -12825.176} C_VEL
LIN {X 0,Y 368.886,Z 274.159,A -85,B 0,C 180,E1 -12828.178,E2 -12828.178} C_VEL
LIN {X 0,Y 368.911,Z 274.156,A -85,B 0,C 180,E1 -12831.36,E2 -12831.36} C_VEL
LIN {X 0,Y 368.939,Z 274.153,A -85,B 0,C 180,E1 -12835.147,E2 -12835.147} C_VEL
LIN {X 0,Y 368.932,Z 274.155,A -85,B 0,C 180,E1 -12839.047,E2 -12839.047} C_VEL
LIN {X 0,Y 368.966,Z 274.151,A -85,B 0,C 180,E1 -12842.797,E2 -12842.797} C_VEL
LIN {X 0,Y 368.936,Z 274.154,A -85,B 0,C 180,E1 -12846.117,E2 -12846.117} C_VEL
LIN {X 0,Y 368.94,Z 274.153,A -85,B 0,C 180,E1 -12849.947,E2 -12849.947} C_VEL
LIN {X 0,Y 368.979,Z 274.146,A -85,B 0,C 180,E1 -12853.399,E2 -12853.399} C_VEL
LIN {X 0,Y 369.061,Z 274.137,A -85,B 0,C 180,E1 -12856.79,E2 -12856.79} C_VEL
LIN {X 0,Y 369.07,Z 274.139,A -85,B 0,C 180,E1 -12860.132,E2 -12860.132} C_VEL
LIN {X 0,Y 369.163,Z 274.124,A -85,B 0,C 180,E1 -12863.441,E2 -12863.441} C_VEL
LIN {X 0,Y 369.312,Z 274.109,A -85,B 0,C 180,E1 -12867.819,E2 -12867.819} C_VEL
LIN {X 0,Y 369.456,Z 274.091,A -85,B 0,C 180,E1 -12870,E2 -12870} C_VEL
LIN {X 0,Y 369.317,Z 274.107,A -85,B 0,C 180,E1 -12872.181,E2 -12872.181} C_VEL
LIN {X 0,Y 369.177,Z 274.122,A -85,B 0,C 180,E1 -12876.559,E2 -12876.559} C_VEL
LIN {X 0,Y 369.066,Z 274.139,A -85,B 0,C 180,E1 -12879.868,E2 -12879.868} C_VEL
LIN {X 0,Y 369.04,Z 274.144,A -85,B 0,C 180,E1 -12883.772,E2 -12883.772} C_VEL
LIN {X 0,Y 369.004,Z 274.147,A -85,B 0,C 180,E1 -12887.768,E2 -12887.768} C_VEL
LIN {X 0,Y 368.932,Z 274.155,A -85,B 0,C 180,E1 -12891.22,E2 -12891.22} C_VEL
LIN {X 0,Y 368.961,Z 274.149,A -85,B 0,C 180,E1 -12894.775,E2 -12894.775} C_VEL
LIN {X 0,Y 368.966,Z 274.152,A -85,B 0,C 180,E1 -12897.203,E2 -12897.203} C_VEL
LIN {X 0,Y 368.932,Z 274.155,A -85,B 0,C 180,E1 -12900.954,E2 -12900.954} C_VEL
LIN {X 0,Y 368.932,Z 274.156,A -85,B 0,C 180,E1 -12905.001,E2 -12905.001} C_VEL
LIN {X 0,Y 368.88,Z 274.16,A -85,B 0,C 180,E1 -12908.634,E2 -12908.634} C_VEL
LIN {X 0,Y 368.877,Z 274.163,A -85,B 0,C 180,E1 -12908.947,E2 -12908.947} C_VEL
LIN {X 0,Y 368.215,Z 274.252,A -85,B 0,C 180,E1 -12909.858,E2 -12909.858} C_VEL
LIN {X 0,Y 365.342,Z 274.607,A -85,B 0,C 180,E1 -12911.339,E2 -12911.339} C_VEL
LIN {X 0,Y 362.911,Z 274.904,A -85,B 0,C 180,E1 -12912.537,E2 -12912.537} C_VEL
LIN {X 0,Y 361.882,Z 275.032,A -85,B 0,C 180,E1 -12913.464,E2 -12913.464} C_VEL
LIN {X 0,Y 361.807,Z 275.038,A -85,B 0,C 180,E1 -12913.778,E2 -12913.778} C_VEL
LIN {X 0,Y 361.839,Z 275.036,A -85,B 0,C 180,E1 -12917.568,E2 -12917.568} C_VEL
LIN {X 0,Y 361.874,Z 275.035,A -85,B 0,C 180,E1 -12920.973,E2 -12920.973} C_VEL
LIN {X 0,Y 361.878,Z 275.035,A -85,B 0,C 180,E1 -12924.655,E2 -12924.655} C_VEL
LIN {X 0,Y 361.842,Z 275.038,A -85,B 0,C 180,E1 -12928.371,E2 -12928.371} C_VEL
LIN {X 0,Y 361.912,Z 275.029,A -85,B 0,C 180,E1 -12932.221,E2 -12932.221} C_VEL
LIN {X 0,Y 361.93,Z 275.028,A -85,B 0,C 180,E1 -12934.71,E2 -12934.71} C_VEL
LIN {X 0,Y 361.865,Z 275.036,A -85,B 0,C 180,E1 -12938.345,E2 -12938.345} C_VEL
LIN {X 0,Y 361.971,Z 275.022,A -85,B 0,C 180,E1 -12942.061,E2 -12942.061} C_VEL
LIN {X 0,Y 362.002,Z 275.019,A -85,B 0,C 180,E1 -12946.101,E2 -12946.101} C_VEL
LIN {X 0,Y 362.004,Z 275.018,A -85,B 0,C 180,E1 -12949.937,E2 -12949.937} C_VEL
LIN {X 0,Y 362.127,Z 275,A -85,B 0,C 180,E1 -12953.313,E2 -12953.313} C_VEL
LIN {X 0,Y 362.282,Z 274.984,A -85,B 0,C 180,E1 -12957.776,E2 -12957.776} C_VEL
LIN {X 0,Y 362.384,Z 274.972,A -85,B 0,C 180,E1 -12960,E2 -12960} C_VEL
LIN {X 0,Y 362.284,Z 274.983,A -85,B 0,C 180,E1 -12962.223,E2 -12962.223} C_VEL
LIN {X 0,Y 362.129,Z 274.999,A -85,B 0,C 180,E1 -12966.687,E2 -12966.687} C_VEL
LIN {X 0,Y 362.003,Z 275.019,A -85,B 0,C 180,E1 -12970.063,E2 -12970.063} C_VEL
LIN {X 0,Y 362.001,Z 275.019,A -85,B 0,C 180,E1 -12973.899,E2 -12973.899} C_VEL
LIN {X 0,Y 361.97,Z 275.022,A -85,B 0,C 180,E1 -12977.938,E2 -12977.938} C_VEL
LIN {X 0,Y 361.896,Z 275.033,A -85,B 0,C 180,E1 -12981.652,E2 -12981.652} C_VEL
LIN {X 0,Y 361.887,Z 275.034,A -85,B 0,C 180,E1 -12985.293,E2 -12985.293} C_VEL
LIN {X 0,Y 361.857,Z 275.037,A -85,B 0,C 180,E1 -12989.073,E2 -12989.073} C_VEL
LIN {X 0,Y 361.85,Z 275.038,A -85,B 0,C 180,E1 -12992.944,E2 -12992.944} C_VEL
LIN {X 0,Y 361.909,Z 275.146,A -85,B 0,C 180,E1 -12993.767,E2 -12993.767} C_VEL
LIN {X 0,Y 362.739,Z 279.954,A -85,B 0,C 180,E1 -12997.404,E2 -12997.404} C_VEL
LIN {X 0,Y 363.654,Z 285.148,A -85,B 0,C 180,E1 -13001.086,E2 -13001.086} C_VEL
LIN {X 0,Y 364.606,Z 290.26,A -85,B 0,C 180,E1 -13004.504,E2 -13004.504} C_VEL
LIN {X 0,Y 365.205,Z 294.188,A -85,B 0,C 180,E1 -13006.993,E2 -13006.993} C_VEL
LIN {X 0,Y 365.118,Z 297.761,A -85,B 0,C 180,E1 -13009.122,E2 -13009.122} C_VEL
LIN {X 0,Y 364.499,Z 303.251,A -85,B 0,C 180,E1 -13012.235,E2 -13012.235} C_VEL
LIN {X 0,Y 363.862,Z 308.781,A -85,B 0,C 180,E1 -13015.264,E2 -13015.264} C_VEL
LIN {X 0,Y 363.189,Z 314.876,A -85,B 0,C 180,E1 -13018.501,E2 -13018.501} C_VEL
LIN {X 0,Y 362.617,Z 320.728,A -85,B 0,C 180,E1 -13021.53,E2 -13021.53} C_VEL
LIN {X 0,Y 367.422,Z 339.515,A -85,B 0,C 180,E1 -13022.576,E2 -13022.576} C_VEL
LIN {X 0,Y 371.148,Z 355.857,A -85,B 0,C 180,E1 -13023.683,E2 -13023.683} C_VEL
LIN {X 0,Y 373.325,Z 368.216,A -85,B 0,C 180,E1 -13024.638,E2 -13024.638} C_VEL
LIN {X 0,Y 371.829,Z 382.667,A -85,B 0,C 180,E1 -13025.726,E2 -13025.726} C_VEL
LIN {X 0,Y 369.949,Z 395.844,A -85,B 0,C 180,E1 -13026.932,E2 -13026.932} C_VEL
LIN {X 0,Y 368.117,Z 409.268,A -85,B 0,C 180,E1 -13028.437,E2 -13028.437} C_VEL
LIN {X 0,Y 366.361,Z 421.18,A -85,B 0,C 180,E1 -13030.048,E2 -13030.048} C_VEL
LIN {X 0,Y 364.893,Z 431.762,A -85,B 0,C 180,E1 -13031.761,E2 -13031.761} C_VEL
LIN {X 0,Y 363.431,Z 441.889,A -85,B 0,C 180,E1 -13033.716,E2 -13033.716} C_VEL
LIN {X 0,Y 362.246,Z 450.908,A -85,B 0,C 180,E1 -13035.824,E2 -13035.824} C_VEL
LIN {X 0,Y 361.542,Z 457.369,A -85,B 0,C 180,E1 -13037.653,E2 -13037.653} C_VEL
LIN {X 0,Y 360.879,Z 463.877,A -85,B 0,C 180,E1 -13039.905,E2 -13039.905} C_VEL
LIN {X 0,Y 360.574,Z 468.931,A -85,B 0,C 180,E1 -13042.158,E2 -13042.158} C_VEL
LIN {X 0,Y 360.394,Z 472.637,A -85,B 0,C 180,E1 -13044.404,E2 -13044.404} C_VEL
LIN {X 0,Y 360.323,Z 475.072,A -85,B 0,C 180,E1 -13046.645,E2 -13046.645} C_VEL
LIN {X 0,Y 360.453,Z 476.271,A -85,B 0,C 180,E1 -13048.883,E2 -13048.883} C_VEL
LIN {X 0,Y 360.455,Z 476.211,A -85,B 0,C 180,E1 -13051.117,E2 -13051.117} C_VEL
LIN {X 0,Y 360.335,Z 474.938,A -85,B 0,C 180,E1 -13053.354,E2 -13053.354} C_VEL
LIN {X 0,Y 360.427,Z 472.461,A -85,B 0,C 180,E1 -13055.595,E2 -13055.595} C_VEL
LIN {X 0,Y 360.583,Z 468.735,A -85,B 0,C 180,E1 -13057.842,E2 -13057.842} C_VEL
LIN {X 0,Y 360.877,Z 463.69,A -85,B 0,C 180,E1 -13060.095,E2 -13060.095} C_VEL
LIN {X 0,Y 361.54,Z 457.228,A -85,B 0,C 180,E1 -13062.347,E2 -13062.347} C_VEL
LIN {X 0,Y 362.482,Z 449.205,A -85,B 0,C 180,E1 -13064.599,E2 -13064.599} C_VEL
LIN {X 0,Y 363.811,Z 439.439,A -85,B 0,C 180,E1 -13066.844,E2 -13066.844} C_VEL
LIN {X 0,Y 365.381,Z 429.262,A -85,B 0,C 180,E1 -13068.795,E2 -13068.795} C_VEL
LIN {X 0,Y 366.981,Z 419.096,A -85,B 0,C 180,E1 -13070.457,E2 -13070.457} C_VEL
LIN {X 0,Y 369.106,Z 406.227,A -85,B 0,C 180,E1 -13072.237,E2 -13072.237} C_VEL
LIN {X 0,Y 371.499,Z 392.143,A -85,B 0,C 180,E1 -13073.852,E2 -13073.852} C_VEL
LIN {X 0,Y 373.675,Z 379.04,A -85,B 0,C 180,E1 -13075.114,E2 -13075.114} C_VEL
LIN {X 0,Y 375.024,Z 369.61,A -85,B 0,C 180,E1 -13075.904,E2 -13075.904} C_VEL
LIN {X 0,Y 373.261,Z 350.225,A -85,B 0,C 180,E1 -13077.755,E2 -13077.755} C_VEL
LIN {X 0,Y 371.565,Z 340.014,A -85,B 0,C 180,E1 -13078.725,E2 -13078.725} C_VEL
LIN {X 0,Y 368.442,Z 327.909,A -85,B 0,C 180,E1 -13080.004,E2 -13080.004} C_VEL
LIN {X 0,Y 366.292,Z 321.85,A -85,B 0,C 180,E1 -13080.739,E2 -13080.739} C_VEL
LIN {X 0,Y 364.877,Z 317.631,A -85,B 0,C 180,E1 -13081.262,E2 -13081.262} C_VEL
LIN {X 0,Y 363.313,Z 313.915,A -85,B 0,C 180,E1 -13081.793,E2 -13081.793} C_VEL
LIN {X 0,Y 363.042,Z 312.329,A -85,B 0,C 180,E1 -13081.981,E2 -13081.981} C_VEL
LIN {X 0,Y 363.813,Z 306.773,A -85,B 0,C 180,E1 -13085.418,E2 -13085.418} C_VEL
LIN {X 0,Y 364.484,Z 302.939,A -85,B 0,C 180,E1 -13088.1,E2 -13088.1} C_VEL
LIN {X 0,Y 365.3,Z 298.954,A -85,B 0,C 180,E1 -13091.382,E2 -13091.382} C_VEL
LIN {X 0,Y 365.464,Z 296.646,A -85,B 0,C 180,E1 -13093.812,E2 -13093.812} C_VEL
LIN {X 0,Y 365.235,Z 294.973,A -85,B 0,C 180,E1 -13096.154,E2 -13096.154} C_VEL
LIN {X 0,Y 364.623,Z 293.617,A -85,B 0,C 180,E1 -13099.055,E2 -13099.055} C_VEL
LIN {X 0,Y 363.91,Z 292.854,A -85,B 0,C 180,E1 -13102.356,E2 -13102.356} C_VEL
LIN {X 0,Y 363.534,Z 292.83,A -85,B 0,C 180,E1 -13104.59,E2 -13104.59} C_VEL
LIN {X 0,Y 364.677,Z 295.514,A -85,B 0,C 180,E1 -13105.055,E2 -13105.055} C_VEL
LIN {X 0,Y 366.344,Z 297.505,A -85,B 0,C 180,E1 -13105.547,E2 -13105.547} C_VEL
LIN {X 0,Y 371.681,Z 306.787,A -85,B 0,C 180,E1 -13107.221,E2 -13107.221} C_VEL
LIN {X 0,Y 375.709,Z 315.443,A -85,B 0,C 180,E1 -13108.532,E2 -13108.532} C_VEL
LIN {X 0,Y 378.347,Z 323.382,A -85,B 0,C 180,E1 -13109.564,E2 -13109.564} C_VEL
LIN {X 0,Y 378.321,Z 326.334,A -85,B 0,C 180,E1 -13109.813,E2 -13109.813} C_VEL
LIN {X 0,Y 376.239,Z 340.601,A -85,B 0,C 180,E1 -13110.944,E2 -13110.944} C_VEL
LIN {X 0,Y 373.763,Z 356.241,A -85,B 0,C 180,E1 -13112.47,E2 -13112.47} C_VEL
LIN {X 0,Y 371.707,Z 368.511,A -85,B 0,C 180,E1 -13113.922,E2 -13113.922} C_VEL
LIN {X 0,Y 369.735,Z 379.753,A -85,B 0,C 180,E1 -13115.484,E2 -13115.484} C_VEL
LIN {X 0,Y 367.873,Z 390.333,A -85,B 0,C 180,E1 -13117.241,E2 -13117.241} C_VEL
LIN {X 0,Y 366.119,Z 400.212,A -85,B 0,C 180,E1 -13119.199,E2 -13119.199} C_VEL
LIN {X 0,Y 364.427,Z 409.533,A -85,B 0,C 180,E1 -13121.452,E2 -13121.452} C_VEL
LIN {X 0,Y 363.157,Z 416.94,A -85,B 0,C 180,E1 -13123.704,E2 -13123.704} C_VEL
LIN {X 0,Y 362.226,Z 422.749,A -85,B 0,C 180,E1 -13125.958,E2 -13125.958} C_VEL
LIN {X 0,Y 361.675,Z 426.141,A -85,B 0,C 180,E1 -13127.658,E2 -13127.658} C_VEL
LIN {X 0,Y 361.116,Z 429.486,A -85,B 0,C 180,E1 -13129.912,E2 -13129.912} C_VEL
LIN {X 0,Y 360.833,Z 431.55,A -85,B 0,C 180,E1 -13132.164,E2 -13132.164} C_VEL
LIN {X 0,Y 360.707,Z 432.368,A -85,B 0,C 180,E1 -13134.41,E2 -13134.41} C_VEL
LIN {X 0,Y 360.633,Z 431.957,A -85,B 0,C 180,E1 -13136.649,E2 -13136.649} C_VEL
LIN {X 0,Y 360.597,Z 430.32,A -85,B 0,C 180,E1 -13138.884,E2 -13138.884} C_VEL
LIN {X 0,Y 360.638,Z 427.409,A -85,B 0,C 180,E1 -13141.117,E2 -13141.117} C_VEL
LIN {X 0,Y 361.017,Z 423.177,A -85,B 0,C 180,E1 -13143.348,E2 -13143.348} C_VEL
LIN {X 0,Y 361.427,Z 419.095,A -85,B 0,C 180,E1 -13145.02,E2 -13145.02} C_VEL
LIN {X 0,Y 361.81,Z 412.371,A -85,B 0,C 180,E1 -13147.254,E2 -13147.254} C_VEL
LIN {X 0,Y 362.632,Z 403.964,A -85,B 0,C 180,E1 -13149.482,E2 -13149.482} C_VEL
LIN {X 0,Y 363.671,Z 395.022,A -85,B 0,C 180,E1 -13151.425,E2 -13151.425} C_VEL
LIN {X 0,Y 364.82,Z 384.321,A -85,B 0,C 180,E1 -13153.366,E2 -13153.366} C_VEL
LIN {X 0,Y 366.081,Z 373.412,A -85,B 0,C 180,E1 -13155.021,E2 -13155.021} C_VEL
LIN {X 0,Y 367.502,Z 360.454,A -85,B 0,C 180,E1 -13156.67,E2 -13156.67} C_VEL
LIN {X 0,Y 368.793,Z 347.545,A -85,B 0,C 180,E1 -13158.04,E2 -13158.04} C_VEL
LIN {X 0,Y 370.236,Z 333.588,A -85,B 0,C 180,E1 -13159.258,E2 -13159.258} C_VEL
LIN {X 0,Y 371.435,Z 318.724,A -85,B 0,C 180,E1 -13160.316,E2 -13160.316} C_VEL
LIN {X 0,Y 371.47,Z 315.539,A -85,B 0,C 180,E1 -13160.524,E2 -13160.524} C_VEL
LIN {X 0,Y 367.353,Z 300.288,A -85,B 0,C 180,E1 -13161.611,E2 -13161.611} C_VEL
LIN {X 0,Y 362.763,Z 285.107,A -85,B 0,C 180,E1 -13162.528,E2 -13162.528} C_VEL
LIN {X 0,Y 360.963,Z 278.848,A -85,B 0,C 180,E1 -13162.868,E2 -13162.868} C_VEL
LIN {X 0,Y 361.006,Z 275.461,A -85,B 0,C 180,E1 -13166.6,E2 -13166.6} C_VEL
LIN {X 0,Y 361.273,Z 275.111,A -85,B 0,C 180,E1 -13169.1,E2 -13169.1} C_VEL
LIN {X 0,Y 361.518,Z 275.078,A -85,B 0,C 180,E1 -13171.661,E2 -13171.661} C_VEL
LIN {X 0,Y 361.741,Z 275.048,A -85,B 0,C 180,E1 -13174.293,E2 -13174.293} C_VEL
LIN {X 0,Y 361.86,Z 275.037,A -85,B 0,C 180,E1 -13177.222,E2 -13177.222} C_VEL
LIN {X 0,Y 361.837,Z 275.039,A -85,B 0,C 180,E1 -13180.755,E2 -13180.755} C_VEL
LIN {X 0,Y 361.82,Z 275.038,A -85,B 0,C 180,E1 -13184.369,E2 -13184.369} C_VEL
LIN {X 0,Y 361.839,Z 275.036,A -85,B 0,C 180,E1 -13187.568,E2 -13187.568} C_VEL
LIN {X 0,Y 361.872,Z 275.035,A -85,B 0,C 180,E1 -13190.974,E2 -13190.974} C_VEL
LIN {X 0,Y 361.877,Z 275.035,A -85,B 0,C 180,E1 -13194.655,E2 -13194.655} C_VEL
LIN {X 0,Y 361.841,Z 275.038,A -85,B 0,C 180,E1 -13198.371,E2 -13198.371} C_VEL
LIN {X 0,Y 361.911,Z 275.03,A -85,B 0,C 180,E1 -13202.221,E2 -13202.221} C_VEL
LIN {X 0,Y 361.929,Z 275.028,A -85,B 0,C 180,E1 -13204.71,E2 -13204.71} C_VEL
LIN {X 0,Y 361.868,Z 275.035,A -85,B 0,C 180,E1 -13208.786,E2 -13208.786} C_VEL
LIN {X 0,Y 361.971,Z 275.022,A -85,B 0,C 180,E1 -13212.061,E2 -13212.061} C_VEL
LIN {X 0,Y 362.001,Z 275.019,A -85,B 0,C 180,E1 -13216.101,E2 -13216.101} C_VEL
LIN {X 0,Y 362.034,Z 275.015,A -85,B 0,C 180,E1 -13219.938,E2 -13219.938} C_VEL
LIN {X 0,Y 362.126,Z 275,A -85,B 0,C 180,E1 -13223.313,E2 -13223.313} C_VEL
LIN {X 0,Y 362.275,Z 274.985,A -85,B 0,C 180,E1 -13227.776,E2 -13227.776} C_VEL
LIN {X 0,Y 362.405,Z 274.97,A -85,B 0,C 180,E1 -13230,E2 -13230} C_VEL
LIN {X 0,Y 362.281,Z 274.983,A -85,B 0,C 180,E1 -13232.224,E2 -13232.224} C_VEL
LIN {X 0,Y 362.138,Z 274.998,A -85,B 0,C 180,E1 -13236.687,E2 -13236.687} C_VEL
LIN {X 0,Y 362.003,Z 275.018,A -85,B 0,C 180,E1 -13240.063,E2 -13240.063} C_VEL
LIN {X 0,Y 362.001,Z 275.019,A -85,B 0,C 180,E1 -13243.899,E2 -13243.899} C_VEL
LIN {X 0,Y 361.971,Z 275.022,A -85,B 0,C 180,E1 -13247.939,E2 -13247.939} C_VEL
LIN {X 0,Y 361.895,Z 275.032,A -85,B 0,C 180,E1 -13251.653,E2 -13251.653} C_VEL
LIN {X 0,Y 361.932,Z 275.029,A -85,B 0,C 180,E1 -13255.29,E2 -13255.29} C_VEL
LIN {X 0,Y 361.912,Z 275.028,A -85,B 0,C 180,E1 -13257.779,E2 -13257.779} C_VEL
LIN {X 0,Y 361.841,Z 275.038,A -85,B 0,C 180,E1 -13261.629,E2 -13261.629} C_VEL
LIN {X 0,Y 361.877,Z 275.035,A -85,B 0,C 180,E1 -13265.345,E2 -13265.345} C_VEL
LIN {X 0,Y 361.829,Z 275.041,A -85,B 0,C 180,E1 -13269.018,E2 -13269.018} C_VEL
LIN {X 0,Y 361.835,Z 275.04,A -85,B 0,C 180,E1 -13272.829,E2 -13272.829} C_VEL
LIN {X 0,Y 361.807,Z 275.038,A -85,B 0,C 180,E1 -13273.778,E2 -13273.778} C_VEL
LIN {X 0,Y 361.155,Z 275.124,A -85,B 0,C 180,E1 -13274.707,E2 -13274.707} C_VEL
LIN {X 0,Y 358.29,Z 275.478,A -85,B 0,C 180,E1 -13276.218,E2 -13276.218} C_VEL
LIN {X 0,Y 355.869,Z 275.781,A -85,B 0,C 180,E1 -13277.441,E2 -13277.441} C_VEL
LIN {X 0,Y 354.854,Z 275.907,A -85,B 0,C 180,E1 -13278.388,E2 -13278.388} C_VEL
LIN {X 0,Y 354.785,Z 275.917,A -85,B 0,C 180,E1 -13278.708,E2 -13278.708} C_VEL
LIN {X 0,Y 354.81,Z 275.912,A -85,B 0,C 180,E1 -13282.117,E2 -13282.117} C_VEL
LIN {X 0,Y 354.816,Z 275.914,A -85,B 0,C 180,E1 -13284.941,E2 -13284.941} C_VEL
LIN {X 0,Y 354.797,Z 275.916,A -85,B 0,C 180,E1 -13288.405,E2 -13288.405} C_VEL
